//(7,95) Przesuwanie formatek sprzed 
rtfbLidSealerDrag(CLK:=P06_LidSealer.fbLidSealerDragStation.eRunningState = E_DragStationState.eDraging AND P06_LidSealer.fbLidSealerDragStation.lrActualDragPosition>80);
IF rtfbLidSealerDrag.Q THEN
	eLidSealerPackageState[1]			:=	eBeforeLidSealerPackageState[1];
	eBeforeLidSealerPackageState[1]		:=	eClearPackageState;
	eLidSealerPackageState[2]			:=	eBeforeLidSealerPackageState[2];
	eBeforeLidSealerPackageState[2]		:=	eClearPackageState;
END_IF
		
//(7,96) 
fbIbLidFeederAfterSensor 	(bIN:= 	IbLidFeederAfterSensor ,	tFilterTimeOn:=T#40MS,	tFilterTimeOff:=T#20MS); //BYŁO 20ms
ftfbIbLidFeederAfterSensor	(CLK:=	fbIbLidFeederAfterSensor.bOUT);
rtfbIbLidFeederAfterSensor	(CLK:=	fbIbLidFeederAfterSensor.bOUT);
fbMRAfterLidFeederPackageState(
						bFirstCycle:= GVL.bFirstCycle,
						bTrigger:=ftfbIbLidFeederAfterSensor.Q,
						tTriggerFilterTimeOn:=T#0MS,
						tTriggerFilterTimeOff:=T#0MS,
						bTriggerBottle:=FALSE,
						bWithBottleControl:=FALSE,
						bWithCapControl:=FALSE,
						bWithFormControlTrigerCounter:=FALSE,
						bMoveOnlyToLastExitRegister:=FALSE,
						bRotateEntranceRegisterBefore:=FALSE,
						bNoKeepTryingMove:=TRUE,
						bTriggerCap:=FALSE,
						bReset:=bResetStates,
						iEntranceArrayElements:=2,
						iExitArrayElements:=2,
						bInvertWriting:=FALSE,
						eClearPackageState:=eClearPackageState,
						bTriggerCounter:=bMRCapCorrect,
						eEntranceState:=eAfterLidFeederPackageState,
						eExitState:=eBeforeLidSealerPackageState,
						bKeepTryingMove:=bKeepTryingMove796,
						bError=>,
						iError=>,
						bTriggerDone=>,
						bTriggerFilteredOUT=>);			

// (7,97) Przesuwanie formatek spod zakrecearek za zakrecarki  
rtfbLidFeederDrag(CLK:=
						(P06_LidFeeder.fbLidFeederDragStation.eRunningState = E_DragStationState.eDraging AND P06_LidFeeder.fbLidFeederDragStation.lrActualDragPosition>80) OR
						(P06_WickFeeder.fbWickFeederDragStation.eRunningState = E_DragStationState.eDraging AND P06_WickFeeder.fbWickFeederDragStation.lrActualDragPosition>80)
						);
IF rtfbLidFeederDrag.Q THEN
	eAfterLidFeederPackageState[1]		:=	eLidFeederPackageState[1];
	eAfterLidFeederPackageState[2]		:=	eLidFeederPackageState[2];
	eLidFeederPackageState[1]			:=	eClearPackageState;
	eLidFeederPackageState[2]			:=	eClearPackageState;
END_IF

//(7,98) Przesuwanie formatek sprzed sprawdzania platynek na platynki
IF rtfbLidFeederDrag.Q THEN
	eLidFeederPackageState[1]			:=	eBeforeLidFeederPackageState[1];
	eBeforeLidFeederPackageState[1]		:=	eClearPackageState;
	eLidFeederPackageState[2]			:=	eBeforeLidFeederPackageState[2];
	eBeforeLidFeederPackageState[2]		:=	eClearPackageState;
END_IF

//(7,99)
fbIbLidFeederThirdFormSensor				(bIN:= 	IbLidFeederThirdFormSensor,					tFilterTimeOn:=T#30MS,	tFilterTimeOff:=T#30MS); 
ftfbIbLidFeederThirdFormSensor				(CLK:=	fbIbLidFeederThirdFormSensor.bOUT, 			Q=>); 
rtfbIbLidFeederThirdFormSensor				(CLK:=	fbIbLidFeederThirdFormSensor.bOUT, 			Q=>);
ftbMRBeforeLidFeeder2Block					(CLK:=	bMRBeforeLidFeeder2Block,					Q=>);
tofftbMRBeforeLidFeeder2Block				(IN:=	ftbMRBeforeLidFeeder2Block.Q,				PT:=T#1100MS);	
// Ustawianie blokady dla ruchu tylko w jedną stronę siłownika
IF ((P06_LidFeeder.fbLidFeederDragStation.eRunningState = E_DragStationState.eDraging)OR (P06_WickFeeder.fbWickFeederDragStation.eRunningState = E_DragStationState.eDraging))
	AND NOT bMRBeforeLidFeeder2Block AND NOT tofftbMRBeforeLidFeeder2Block.Q THEN
	bMRBeforeLidFeeder2Block := TRUE;
END_IF
IF bMRBeforeLidFeeder2Block AND 
	(
	(P06_LidFeeder.fbLidFeederDragStation.eRunningState = E_DragStationState.eDraging AND P06_LidFeeder.fbLidFeederDragStation.lrActualDragPosition>90) OR
	(P06_WickFeeder.fbWickFeederDragStation.eRunningState = E_DragStationState.eDraging AND P06_WickFeeder.fbWickFeederDragStation.lrActualDragPosition>90)
	)
 THEN	
	bMRBeforeLidFeeder2Block := FALSE;
END_IF

fbMRBeforeLidFeeder2PackageState(
                        bFirstCycle:= GVL.bFirstCycle,
                        bTrigger:=rtfbIbLidFeederThirdFormSensor.Q AND NOT bMRBeforeLidFeeder2Block,
                        tTriggerFilterTimeOn:=T#0MS,
                        tTriggerFilterTimeOff:=T#0MS,
                        bTriggerBottle:=FALSE,
                        bWithBottleControl:=FALSE,
                        bWithCapControl:=FALSE,
                        bWithFormControlTrigerCounter:=FALSE,
                        bRotateEntranceRegisterBefore:=FALSE,
                        bNoKeepTryingMove:=TRUE,
                        bTriggerCap:=,
                        bReset:=bResetStates,
                        iEntranceArrayElements:=4,
                        iExitArrayElements:=2,
                        bInvertWriting:=FALSE,
                        eClearPackageState:=eClearPackageState,
                        bTriggerCounter:=bMRLidFeederFormInCap,
                        eEntranceState:=eBeforeLidFeeder2PackageState,
                        eExitState:=eBeforeLidFeederPackageState,
                        bKeepTryingMove:=bKeepTryingMove799,
                        bError=>,
                        iError=>,
                        bTriggerDone=>,
                        bTriggerFilteredOUT=>); 
IF fbMRBeforeLidFeeder2PackageState.bTrigger THEN iLFTest1:=iLFTest1+1; END_IF 
// (7,99) A - Dodatkowe przesuniecie na zboczne narastajace
//IF rtfbIbLidFeederThirdFormSensor.Q AND NOT eBeforeLidFeeder2PackageState[1].bFormPresent THEN
//	eBeforeLidFeeder2PackageState[1] := eBeforeLidFeeder2PackageState[2];
//	eBeforeLidFeeder2PackageState[2] := eClearPackageState;
//	eBeforeLidFeeder2PackageState[2] := eBeforeLidFeeder2PackageState[3];
//	eBeforeLidFeeder2PackageState[3] := eClearPackageState;	
//	eBeforeLidFeeder2PackageState[3] := eBeforeLidFeeder2PackageState[4];
//	eBeforeLidFeeder2PackageState[4] := eClearPackageState;			
//END_IF


// (8) Przesuwanie formatek z wagi w kosmos	LidFeeder		
fbIbWeight1FormSensor			(bIN:= 	P05_Weight.IbWeight1FormSensor,		tFilterTimeOn:=T#40MS,	tFilterTimeOff:=T#40MS);
ftfbIbWeight1FormSensor			(CLK:=	fbIbWeight1FormSensor.bOUT, 		Q=>);	

fbMRAfterWeightPackageStateLF(		///ZMIANAAAA
						bFirstCycle:= GVL.bFirstCycle,
						bTrigger:=ftfbIbWeight1FormSensor.Q,
						tTriggerFilterTimeOn:=T#0MS,
						tTriggerFilterTimeOff:=T#0MS,
						bTriggerBottle:=FALSE,
						bWithBottleControl:=FALSE,
						bWithCapControl:=FALSE,
						bWithFormControlTrigerCounter:=FALSE,
						bMoveOnlyToLastExitRegister:=FALSE,
						bRotateEntranceRegisterBefore:=FALSE,
						bNoKeepTryingMove:=FALSE,
						bTriggerCap:=FALSE,
						bReset:=bResetStates,
						iEntranceArrayElements:=4,
						iExitArrayElements:=4,
						bInvertWriting:=FALSE,
						eClearPackageState:=eClearPackageState,
						bTriggerCounter:=bMRFormExitWeight,
						eEntranceState:=eWeightPackageState,
						eExitState:=eBeforeLidFeeder2PackageState,
						bKeepTryingMove:=bKeepTryingMove4,
						bError=>,
						iError=>,
						bTriggerDone=>,
						bTriggerFilteredOUT=>);				
											
						
// (9) Przesuwanie formatek zza dozownikow na wage
fbIbWeight4FormSensor			(bIN:= 	P05_Weight.IbWeight4FormSensor,		tFilterTimeOn:=T#40MS,	tFilterTimeOff:=T#40MS); //BYLO 20 I 20
//fbIbWeight4FormSensor			(bIN:= 	P00_ReadRFIDCard.bReadedCardAfterDispencers,		tFilterTimeOn:=T#40MS,	tFilterTimeOff:=T#40MS); //BYLO 20 I 20
ftIbWeight4FormSensor			(CLK:=	fbIbWeight4FormSensor.bOUT, 		Q=>);	
fbMRWeightPackageState(
						bFirstCycle:= GVL.bFirstCycle,
						bTrigger:=fbIbWeight4FormSensor.bOUT,//P05_Weight.IbWeight4FormSensor, 
						tTriggerFilterTimeOn:=T#100MS,
						tTriggerFilterTimeOff:=T#20MS,
						bTriggerBottle:=FALSE,
						bWithBottleControl:=FALSE,
						bWithCapControl:=FALSE,
						bWithFormControlTrigerCounter:=FALSE,
						bMoveOnlyToLastExitRegister:=FALSE,
						bRotateEntranceRegisterBefore:=FALSE,
						bNoKeepTryingMove:=FALSE,
						bTriggerCap:=FALSE,
						bReset:=bResetStates,
						iEntranceArrayElements:=4,
						iExitArrayElements:=4,
						bInvertWriting:=FALSE,
						eClearPackageState:=eClearPackageState,
						bTriggerCounter:=bTemp,
						eEntranceState:=eAfterDispencersPackageState,
						eExitState:=eWeightPackageState,
						bKeepTryingMove:=bKeepTryingMove5,
						bError=>,
						iError=>,
						bTriggerDone=>,
						bTriggerFilteredOUT=>);		

						
// (10) Przesuwanie z dozownikow za dozowniki
fbMRAfterDispencerPackageState(
						bFirstCycle:= GVL.bFirstCycle,
						//bTrigger:=P02_Dispencers.fbDispencersDragRightStation.lrActualDragPosition>=130,
						bTrigger:=P00_PackML.tonDispencersDragLeftMiddleSensor.Q, {warning 'Przeciaganie - TON zamiast pozycji'}
						tTriggerFilterTimeOn:=T#0MS,
						tTriggerFilterTimeOff:=T#0MS,
						bInvertWriting:=FALSE,
						bTriggerBottle:=FALSE,
						iEntrenceArrayElements:=4,
						iExitArrayElements:=4,
						bWithFormControlTrigerCounter:=FALSE,
						bMoveOnlyIfFormPresent:=FALSE,
						bMoveOnlyToLastExitRegister:=FALSE,
						bMoveOnlyToLastRegister:=FALSE,
						bNoKeepTryingMove:=FALSE,
						bReset:=bResetStates,
						eClearPackageState:=eClearPackageState,
						bRotateEntranceRegisterBefore:=FALSE,
						bTriggerCounter:=bMRFormExitDispencer,
						eEntranceState:=eDispencersPackageState,
						eExitState:=eAfterDispencersPackageState,
						bKeepTryingMove:=bKeepTryingMove6,
						bError=>,
						iError=>,
						bTriggerDone=>,
						bTriggerFilteredOUT=>);	

// (11) Przesuwanie sprzed dozownikow na dozowniki
fbMRDispencerPackageState(
						bFirstCycle:= GVL.bFirstCycle,
						//bTrigger:=P02_Dispencers.fbDispencersDragRightStation.lrActualDragPosition>=130,
						bTrigger:=P00_PackML.tonDispencersDragLeftMiddleSensor.Q, {warning 'Przeciaganie - TON zamiast pozycji'}						
						tTriggerFilterTimeOn:=T#0MS,
						tTriggerFilterTimeOff:=T#0MS,
						bInvertWriting:=FALSE,
						bTriggerBottle:=FALSE,
						iEntrenceArrayElements:=4,
						iExitArrayElements:=4,
						bWithFormControlTrigerCounter:=FALSE,
						bMoveOnlyIfFormPresent:=FALSE,
						bMoveOnlyToLastExitRegister:=FALSE,
						bMoveOnlyToLastRegister:=FALSE,
						bNoKeepTryingMove:=FALSE,
						bReset:=bResetStates,
						eClearPackageState:=eClearPackageState,
						bRotateEntranceRegisterBefore:=FALSE,
						bTriggerCounter:=bMRFormDispencer,
						eEntranceState:=eBeforeDispencersPackageState,
						eExitState:=eDispencersPackageState,
						bKeepTryingMove:=bKeepTryingMove7,
						bError=>,
						iError=>,
						bTriggerDone=>,
						bTriggerFilteredOUT=>);		
					
// (12) Przesuwanie formatek sprzed szlabanu rpzed dozowniki

fbFilteredFormsSensorGate(bIn:=IbFormCheckFormSensor,	tFilterTimeOn:=T#30MS,	tFilterTimeOff:=T#20MS);					
fbMRBeforeDispencersPackageStateNew(
						bFirstCycle:= GVL.bFirstCycle,
						{warning ''}
						bTrigger:=(*fbFilteredFormsSensorGate.bOUT*)bFormatSensor,
						tTriggerFilterTimeOn:=T#0MS,
						tTriggerFilterTimeOff:=T#0MS,
						{warning 'Add filtered value 2023/06/16'}
						bTriggerBottle:=bBottleSensor (*MAIN.IbBottleInFormCheckBottleSensor*) OR VIS.bSimulation,
						bWithBottleControl:=TRUE,
						bWithCapControl:=FALSE,
						bWithFormControlTrigerCounter:=FALSE,
						bMoveOnlyToLastExitRegister:=FALSE,
						bRotateEntranceRegisterBefore:=FALSE,
						bNoKeepTryingMove:=TRUE,
						bTriggerCap:=,
						bReset:=bResetStates,
						iEntranceArrayElements:=1,
						iExitArrayElements:=4,
						bInvertWriting:=FALSE,
						eClearPackageState:=eClearPackageState,
						bTriggerCounter:=bMRFormExitGate1,
						eEntranceState:=eBeforeGatePackageState,
						eExitState:=eBeforeDispencersPackageState,
						bKeepTryingMove:=bKeepTryingMove8,
						bError=>,
						iError=>,
						bTriggerDone=>,
						bTriggerFilteredOUT=>);			
	
// Przesuwanie formatek spod podjanika butelek w kosmos
eTempState2[1]:=eClearPackageState;
eTempState2[2]:=eClearPackageState;
eTempState2[3]:=eClearPackageState;
fbIbBottleFeederFormPresent(bIn:=P01_BottleFeeder.IbBottleFeederFormGateBeforeSensor,	tFilterTimeOn:=T#20MS,	tFilterTimeOff:=T#20MS);					
ftfbIbBottleFeederFormPresent(CLK:=fbIbBottleFeederFormPresent.bOUT);
				
aSetIDBottle();						
						
//Pierwszy cykl, zeby na poczatek nie wykrywalo zbocza opadajacego				
bFirstCycle:=TRUE;		
GVL.bResetStates:=FALSE;


(**** Zapisywanie RFID  ***)

a2RFID();

(**** Koniec zapisywania RFID  ***)
END_ACTION

ACTION aCycleRegister2Phase:
eClearPackageState.nID := 0;
eClearPackageState.nCardNumber:=0;
eClearPackageState.bFormPresent := FALSE;
eClearPackageState.bBottlePresent := FALSE;
eClearPackageState.bDosingTwoPhases := FALSE;
eClearPackageState.nDispencerNr := 0;
eClearPackageState.nDispencerNrSecondPhase := 0;
eClearPackageState.tDispencingTime := T#0MS;
eClearPackageState.tDispencingTimeSecondPhase := T#0MS;
eClearPackageState.lrDoseVolumeSV := 0.0;
eClearPackageState.lrDoseVolumeCV := 0.0;
eClearPackageState.lrDoseVolumeSVSecondPhase := 0.0;
eClearPackageState.lrDoseVolumeCVSecondPhase := 0.0;
eClearPackageState.bDoseAborted := FALSE;
eClearPackageState.bWeighed := FALSE;
eClearPackageState.bWeightAborted:=FALSE;
eClearPackageState.lrWeightSV := 0.0;
eClearPackageState.lrWeightCV := 0.0;
eClearPackageState.lrWeightMeasuredCV := 0.0;
eClearPackageState.lrMinWeightCV:=0.0;
eClearPackageState.lrMaxWeightCV:=0.0;	
eClearPackageState.lrWeightDif:=0.0;			
eClearPackageState.bWeightOK := FALSE;
eClearPackageState.tWeightingTime := T#0MS;
eClearPackageState.bCapPutted := FALSE;
eClearPackageState.bCapChecked := FALSE;
eClearPackageState.bCapOK := FALSE;
eClearPackageState.bCapGripperScrewed := FALSE;
eClearPackageState.bCapGripperScrewAborted := FALSE;
eClearPackageState.tCapGripperScrewingTime := T#0MS;
eClearPackageState.bCapCorrectPutted := FALSE;
eClearPackageState.bCapCorrectChecked := FALSE;
eClearPackageState.bCapCorrectNOK := FALSE;
eClearPackageState.bCapCorrectCapOn:=FALSE;
eClearPackageState.bBottleTransferedToExit := FALSE;
eClearPackageState.bBottleTransferedToLabeler := FALSE;
bAlwaysFalse:=FALSE;

// (1) HISTORIA
fbIbFirstFormCheckFormSensor	(bIN:= 	P13_BottleTransfer.IbFirstFormCheckFormSensor,	tFilterTimeOn:=T#30MS,	tFilterTimeOff:=T#30MS);// bylo 80 i 20
ftfbIbFirstFormCheckFormSensor	(CLK:=	fbIbFirstFormCheckFormSensor.bOUT, 				Q=>);
rtfbIbFirstFormCheckFormSensor	(CLK:=	fbIbFirstFormCheckFormSensor.bOUT,				Q=>);
fbIbSecondFormCheckFormSensor	(bIN:= 	P13_BottleTransfer.IbSecondFormCheckFormSensor,	tFilterTimeOn:=T#30MS,	tFilterTimeOff:=T#30MS);
rtfbIbSecondFormCheckFormSensor	(CLK:=	fbIbSecondFormCheckFormSensor.bOUT, 			Q=>);
ftfbIbSecondFormCheckFormSensor	(CLK:=	fbIbSecondFormCheckFormSensor.bOUT, 			Q=>);


// (0) Kasowanie formatek za robotem
// BOOL ustawiany przy nastepnym ruchu robota
bRFIDClearAfterRobot;					
iRFIDClearNr1AfterRobot;	
iRFIDClearNr2AfterRobot;
rtiBottleTransferCase2(CLK:=P00_PackML.iBottleTransferCase	=	2,		Q=>);
IF	rtiBottleTransferCase2.Q	THEN
	IF P00_PackML.nCounterFormsToLoad = 2 THEN
		iRFIDClearNr1AfterRobot	:=	ULINT_TO_INT(eRobotPackageState[1].nCardNumber);
		iRFIDClearNr2AfterRobot	:=	ULINT_TO_INT(eRobotPackageState[2].nCardNumber);		
	ELSIF P00_PackML.nCounterFormsToLoad = 1 THEN
		iRFIDClearNr1AfterRobot	:=	ULINT_TO_INT(eRobotPackageState[1].nCardNumber);
		iRFIDClearNr2AfterRobot	:=	0;	
	END_IF
END_IF
IF bRFIDClearAfterRobot THEN 
	FOR i:=1 TO 100 DO	
		IF iRFIDClearNr1AfterRobot > 0 THEN	{warning 'tutaj zmienić na dwa FORy i EXITy'}
			IF eRFID[i].nCardNumber = INT_TO_ULINT(iRFIDClearNr1AfterRobot) THEN
				eRFID[i]						:=	eClearPackageState;
				eRFID[i].bFormPresent			:= TRUE; // wprowadzona zmiana do testów 
				iRFIDClearNr1AfterRobot			:= 0;
				iRFIDClearNr1AfterRobotCount	:=	iRFIDClearNr1AfterRobotCount	+	1;
			END_IF
		END_IF
		IF iRFIDClearNr2AfterRobot > 0 THEN
			IF eRFID[i].nCardNumber = INT_TO_ULINT(iRFIDClearNr2AfterRobot) THEN
				eRFID[i]						:=	eClearPackageState;
				eRFID[i].bFormPresent			:= TRUE;  // Wprowadzona zmiana do testów
				iRFIDClearNr2AfterRobot			:= 0;
				
				iRFIDClearNr2AfterRobotCount	:=	iRFIDClearNr2AfterRobotCount	+	1;
			END_IF
		END_IF		
		IF 	iRFIDClearNr1AfterRobot = 0 AND iRFIDClearNr2AfterRobot = 0 THEN
			bRFIDClearAfterRobot	:=	FALSE;
		END_IF
	END_FOR;
END_IF



IF ftfbIbFirstFormCheckFormSensor.Q THEN
	
	FOR i := 999 TO 2 BY -1 DO		
		eHistoryPackageState[i] := eHistoryPackageState[i-1];
	END_FOR		
	
	FOR i:=1 TO 100 DO	
	
		IF eRobotPackageState[1].nCardNumber=eRFID[i].nCardNumber THEN
			eRFID[i]		:=	eRobotPackageState[1];
			EXIT;
		END_IF;
	
	END_FOR;
	
	eHistoryPackageState[1]	:=	eRobotPackageState[1];
	eRobotPackageState[1]	:=	eClearPackageState; // dodane na testy
	nCheckRobotDone			:=	nCheckRobotDone+1;
	
END_IF

IF bResetStates THEN
	eRobotPackageState[1]:=eClearPackageState;
	eRobotPackageState[2]:=eClearPackageState;
	eRobotTempState[1]:=eClearPackageState;// dodane na testy 31.05
END_IF

IF nFormCounter = 1000 OR bResetHistory THEN 
	FOR i := 1 TO 1000 DO
		eHistoryPackageState[i]:=eClearPackageState;
	END_FOR
	
	nFormCounter := 0 ;
	nID := 0;
END_IF


// (2) PRZESUWANIE POD ROBOTEM
IF rtfbIbFirstFormCheckFormSensor.Q THEN
	eRobotPackageState[1]				:= eRobotTempState[1];
	eRobotTempState[1]					:= eClearPackageState;
END_IF

IF  ftfbIbSecondFormCheckFormSensor.Q THEN
	eRobotTempState[1]					:=	eRobotPackageState[2];
	eRobotPackageState[2]				:=	eClearPackageState;
END_IF

IF rtfbIbSecondFormCheckFormSensor.Q THEN
	eRobotPackageState[2].bFormPresent	:=	TRUE;
END_IF

// (3) Przesuwanie formatek zza zakrecarek pod sprwadzanie nakretek
//Przesuwanie formatek spod sprawdzania zakretek na robota
//Usuwanie rejestru bo jest nieuzywant	
//eUnderCorrectCapPackageState[1]			:=	eClearPackageState;	
eUnderCorrectCapPackageState[2]			:=	eClearPackageState;	
eUnderCorrectCapPackageState[3]			:=	eClearPackageState;	
eUnderCorrectCapPackageState[4]			:=	eClearPackageState;	
eUnderCorrectCapPackageState[5]			:=	eClearPackageState;	
eUnderCorrectCapPackageState[6]			:=	eClearPackageState;		
eUnderCorrectCapPackageState[7]			:=	eClearPackageState;		
eUnderCorrectCapPackageState[8]			:=	eClearPackageState;									//bylo 400ms?
fbIbCapCorrectCheckFormSensor			(bIN:= 	P11_CapCorrectCheck.IbCapCorrectCheckFormSensor,	tFilterTimeOn:=T#10MS,	tFilterTimeOff:=T#0MS); //BYŁO 20ms
rtfbIbCapCorrectCheckFormSensor			(CLK:=	fbIbCapCorrectCheckFormSensor.bOUT, 					Q=>); // dd do testów
ftfbIbCapCorrectCheckFormSensor			(CLK:=	fbIbCapCorrectCheckFormSensor.bOUT, 					Q=>);

//Czujnik przesuwania rejestru za zakręcarką
fbIbCapCorrectCheckAfterScrewerFormSensor (bIN:= 	P11_CapCorrectCheck.IbCapCorrectCheckAfterScrewerFormSensor,	tFilterTimeOn:=T#40MS,	tFilterTimeOff:=T#0MS); //BYŁO 20ms
ftfbIbCapCorrectCheckAfterScrewerFormSensor(CLK:=fbIbCapCorrectCheckAfterScrewerFormSensor.bOUT);

IF rtfbIbCapCorrectCheckFormSensor.Q AND NOT eUnderCorrectCapPackageState[1].bFormPresent THEN  			//dd do testów USUNAĆ
	eUnderCorrectCapPackageState[1].bFormPresent  :=	TRUE;  												//dd do testów USUNAĆ
	iTestCCC2	:=	iTestCCC2	+	1;																		//dd do testów USUNAĆ
END_IF  																								

IF 	ftfbIbCapCorrectCheckFormSensor.Q THEN
	eUnderCorrectCapPackageState[1]	:=	eClearPackageState;
	iTestCCC1	:=	iTestCCC1	+	1;
END_IF

fbMRCorrectCapPackageState(
						bFirstCycle:= GVL.bFirstCycle,
						bTrigger:=(*ftfbIbCapCorrectCheckFormSensor.Q*)ftfbIbCapCorrectCheckAfterScrewerFormSensor.Q,
						tTriggerFilterTimeOn:=T#0MS,
						tTriggerFilterTimeOff:=T#0MS,
						bTriggerBottle:=FALSE,
						bWithBottleControl:=FALSE,
						bWithCapControl:=FALSE,
						bWithFormControlTrigerCounter:=FALSE,
						bMoveOnlyToLastExitRegister:=FALSE,
						bRotateEntranceRegisterBefore:=FALSE,
						bNoKeepTryingMove:=TRUE,
						bTriggerCap:=FALSE,
						bReset:=bResetStates,
						iEntranceArrayElements:=2,
						iExitArrayElements:=8,
						bInvertWriting:=FALSE,
						eClearPackageState:=eClearPackageState,
						bTriggerCounter:=bMRCapCorrect,
						eEntranceState:=eAfterScrewerPackageState,
						//eExitState:=eUnderCorrectCapPackageState, //dd do testów USUNAĆ
						eExitState:=eUnderCorrectCapPackageStateTemp,						
						bKeepTryingMove:=bKeepTryingMove1,
						bError=>,
						iError=>,
						bTriggerDone=>,
						bTriggerFilteredOUT=>);			

eUnderCorrectCapPackageStateTemp[1]:= eClearPackageState; //dd do testów USUNAĆ
eUnderCorrectCapPackageStateTemp[2]:= eClearPackageState;//dd do testów USUNAĆ 
						
// (4) Przesuwanie formatek spod zakrecearek za zakrecarki  
//rtfbFormsDragingPneumaticStationDragging(CLK:=P10_GripperScrewer.fbGripperScrewersDragStation.eRunningState = E_DragStationState.eDraging);
rtfbFormsDragingPneumaticStationDragging(CLK:=P10_GripperScrewer.fbGripperScrewersDragStation.eRunningState = E_DragStationState.eDraging AND P10_GripperScrewer.fbGripperScrewersDragStation.lrActualDragPosition>80);

IF rtfbFormsDragingPneumaticStationDragging.Q THEN
	eAfterScrewerPackageState[1]		:=	eUnderScrewerPackageState[1];
	eAfterScrewerPackageState[2]		:=	eUnderScrewerPackageState[2];
	eUnderScrewerPackageState[1]		:=	eClearPackageState;
	eUnderScrewerPackageState[2]		:=	eClearPackageState;
END_IF

								
// (5) Przesuwanie formatek sprzed zakrecarek na zakrecarki
IF rtfbFormsDragingPneumaticStationDragging.Q THEN
	eUnderScrewerPackageState[1]		:=	eBeforeScrewersPackageState[1];
	eBeforeScrewersPackageState[1]		:=	eClearPackageState;
	eUnderScrewerPackageState[2]		:=	eBeforeScrewers2PackageState[1];
	eBeforeScrewers2PackageState[1]		:=	eClearPackageState;
END_IF

// (6) Przesuwanie formatek zza sprawdzania zalozenia na przed zakrecarki
fbIbScrewerThirdFormCheckFormSensor			(bIN:= 	P10_GripperScrewer.IbGripperScrewersThirdFormCheckFormSensor,		tFilterTimeOn:=T#30MS,	tFilterTimeOff:=T#30MS); //BYŁO 20ms
ftfbIbScrewerThirdFormCheckFormSensor		(CLK:=	fbIbScrewerThirdFormCheckFormSensor.bOUT, 			Q=>);
rtfbIbScrewerThirdFormCheckFormSensor		(CLK:=	fbIbScrewerThirdFormCheckFormSensor.bOUT, 			Q=>);
bTrendIbThirdFormCheckFormSensor:=P10_GripperScrewer.IbGripperScrewersThirdFormCheckFormSensor;
bTrendFilteredIbThirdFormCheckFormSensor:=ftfbIbScrewerThirdFormCheckFormSensor.Q;
ftbMRBeforeScrewer2Block 					(CLK:=	bMRBeforeScrewer2Block,								Q=>);
tofftbMRBeforeScrewer2Block					(IN:=	ftbMRBeforeScrewer2Block.Q,							PT:=T#1100MS);//bylo 350		//  bylo 1000			


// Ustawianie blokady dla ruchu tylko w jedną stronę siłownika
IF ( P10_GripperScrewer.fbGripperScrewersDragStation.eRunningState = E_DragStationState.eDraging )
	AND NOT bMRBeforeScrewer2Block AND NOT tofftbMRBeforeScrewer2Block.Q THEN
	bMRBeforeScrewer2Block := TRUE;
END_IF

//IF bMRBeforeScrewer2Block AND P00_PackML.tonGripperScrewerDragMiddleSensor.Q THEN
IF bMRBeforeScrewer2Block AND P10_GripperScrewer.fbGripperScrewersDragStation.eRunningState = E_DragStationState.eDraging AND P10_GripperScrewer.fbGripperScrewersDragStation.lrActualDragPosition>90 THEN	
	bMRBeforeScrewer2Block := FALSE;
END_IF


//(6)
fbMRBeforeScrewer2PackageState(
                        bFirstCycle:= GVL.bFirstCycle,
                        bTrigger:=ftfbIbScrewerThirdFormCheckFormSensor.Q AND NOT bMRBeforeScrewer2Block,
                        tTriggerFilterTimeOn:=T#0MS,
                        tTriggerFilterTimeOff:=T#0MS,
                        bTriggerBottle:=FALSE,
                        bWithBottleControl:=FALSE,
                        bWithCapControl:=FALSE,
                        bWithFormControlTrigerCounter:=FALSE,
                        bRotateEntranceRegisterBefore:=FALSE,
                        bNoKeepTryingMove:=TRUE,
                        bTriggerCap:=,
                        bReset:=bResetStates,
                        iEntranceArrayElements:=2,
                        iExitArrayElements:=2,
                        bInvertWriting:=FALSE,
                        eClearPackageState:=eClearPackageState,
                        bTriggerCounter:=bMRFormInCap,
                        eEntranceState:=eBeforeScrewers2PackageState,
                        eExitState:=eBeforeScrewersPackageState,
                        bKeepTryingMove:=bKeepTryingMove2,
                        bError=>,
                        iError=>,
                        bTriggerDone=>,
                        bTriggerFilteredOUT=>);   										

// (6) A - Dodatkowe przesuniecie na zboczne narastajace
IF rtfbIbScrewerThirdFormCheckFormSensor.Q AND NOT eBeforeScrewers2PackageState[1].bFormPresent THEN
	eBeforeScrewers2PackageState[1] := eBeforeScrewers2PackageState[2];
	eBeforeScrewers2PackageState[2] := eClearPackageState;
END_IF

						
//(7) Przesuwanie formatek spod sprawdzania zalozenia na przed zakrecarki
fbIbCapPuttedCheckFormSensor		(bIN:= 	P09_CapPuttedCheck.IbCapPuttedCheckFormSensor,		tFilterTimeOn:=T#30MS,	tFilterTimeOff:=T#30MS); //Było 20ms
fbIbCapPuttedCheckFormSensorv2		(bIN:= 	P09_CapPuttedCheck.IbCapPuttedCheckFormSensor,		tFilterTimeOn:=T#30MS,	tFilterTimeOff:=T#30MS); //Było 20ms
ftfbIbCapPuttedCheckFormSensor		(CLK:=	fbIbCapPuttedCheckFormSensorv2.bOUT, 					Q=>);

IF ftfbIbCapPuttedCheckFormSensor.Q THEN
	iftfbIbCapPuttedCheckFormSensor := iftfbIbCapPuttedCheckFormSensor+1;
END_IF


bBitTestOn:=TRUE;


fbMRBeforeScrewerPackageState(
                        bFirstCycle:= GVL.bFirstCycle,
                        bTrigger:=ftfbIbCapPuttedCheckFormSensor.Q,
                        tTriggerFilterTimeOn:=T#0MS,
                        tTriggerFilterTimeOff:=T#0MS,
                        bWithCapControl:=TRUE,
                      	bNoKeepTryingMove:=TRUE,
                        bTriggerCap:=P09_CapPuttedCheck.eCapPuttedCheckRunningState = E_CheckerState.eCapOK,
                        bReset:=bResetStates,
                        iEntranceArrayElements:=1,
                        iExitArrayElements:=2,
                        eClearPackageState:=eClearPackageState,
                        eEntranceState:=eBeforeCapControlPackageState,
                        eExitState:=eBeforeScrewers2PackageState,
                        bKeepTryingMove:=bKeepTryingMove3,
						bRFIDReaded:=bRFIDSBeforeScrewerWriteToRegister, // Ustawiany jeżeli Dane z tablicy RFID zostały wpisane do zwykłego rejestru
                        iBottleWithoutCap:=iCapFeederCheckCountNOK,
                        bError=>,
                        iError=>,
                        bTriggerDone=>,
                        bTriggerFilteredOUT=>);   


						
// --------------------------------------

aCycleRegisterROPP();

// (7,5-7,9) Przesuwanie pod sorterem nasadek

aCycleRegisterCapSorter();

// --------------------------------------						
						
// (8) Przesuwanie formatek z wagi w kosmos	

eTempState1[1]:=eClearPackageState;
eTempState1[2]:=eClearPackageState;
eTempState1[3]:=eClearPackageState;
fbIbWeight5FormSensor			(bIN:= 	P05_Weight.IbWeight5FormSensor,		tFilterTimeOn:=T#20MS,	tFilterTimeOff:=T#20MS);
ftfbIbWeight5FormSensor			(CLK:=	fbIbWeight5FormSensor.bOUT, 		Q=>);		
fbMRAfterWeightPackageState(
						bFirstCycle:= GVL.bFirstCycle,
						bTrigger:=ftfbIbWeight5FormSensor.Q,
						tTriggerFilterTimeOn:=T#0MS,
						tTriggerFilterTimeOff:=T#0MS,
						bTriggerBottle:=FALSE,
						bWithBottleControl:=FALSE,
						bWithCapControl:=FALSE,
						bWithFormControlTrigerCounter:=FALSE,
						bMoveOnlyToLastExitRegister:=FALSE,
						bRotateEntranceRegisterBefore:=FALSE,
						bNoKeepTryingMove:=FALSE,
						bTriggerCap:=FALSE,
						bReset:=bResetStates,
						iEntranceArrayElements:=2,
						iExitArrayElements:=4,
						bInvertWriting:=FALSE,
						eClearPackageState:=eClearPackageState,
						bTriggerCounter:=bMRFormExitWeight,
						eEntranceState:=eWeightPackage2PhasePackageState,
						eExitState:=eTempState1,
						bKeepTryingMove:=bKeepTryingMove4,
						bError=>,
						iError=>,
						bTriggerDone=>,
						bTriggerFilteredOUT=>);				

// Przesuwanie formatek dozowników na wagę

fbIbWeight6FormSensor			(bIN:= 	P05_Weight.IbWeight6FormSensor,		tFilterTimeOn:=T#20MS,	tFilterTimeOff:=T#20MS);
ftIbWeight6FormSensor			(CLK:=	fbIbWeight6FormSensor.bOUT, 		Q=>);	
fbMRWeight2PhasePackageState(
						bFirstCycle:= GVL.bFirstCycle,
						bTrigger:=fbIbWeight6FormSensor.bOUT,//P05_Weight.IbWeight6FormSensor, 
						tTriggerFilterTimeOn:=T#100MS,//bylo 50 
						tTriggerFilterTimeOff:=T#20MS,
						bTriggerBottle:=FALSE,
						bWithBottleControl:=FALSE,
						bWithCapControl:=FALSE,
						bWithFormControlTrigerCounter:=FALSE, //bylo true
						bMoveOnlyToLastExitRegister:=FALSE,
						bRotateEntranceRegisterBefore:=FALSE,
						bNoKeepTryingMove:=FALSE,
						bTriggerCap:=FALSE,
						bReset:=bResetStates,
						iEntranceArrayElements:=2,
						iExitArrayElements:=2,
						bInvertWriting:=FALSE,
						eClearPackageState:=eClearPackageState,
						bTriggerCounter:=bTemp,
						eEntranceState:=eAfterDispencer12PackageState2Phase,
						eExitState:=eWeightPackage2PhasePackageState,
						bKeepTryingMove:=bKeepTryingMove15,
						bError=>,
						iError=>,
						bTriggerDone=>,
						bTriggerFilteredOUT=>);		

//Przesuwanie formatek sprzed dozowników 12 ( pierwsze 2 z lewej strony) za dozowniki
						
fbMRAfterDispencer12PackageState(
						bFirstCycle:= GVL.bFirstCycle,
//dp					bTrigger:=P02_Dispencers.fbDispencersDragLeftStation.lrActualDragPosition<=30, // do zmiany 
						bTrigger:=P00_PackML.tonDispencersDragLeftMiddleSensor.Q,
						tTriggerFilterTimeOn:=T#0MS,
						tTriggerFilterTimeOff:=T#0MS,
						bInvertWriting:=FALSE,
						bTriggerBottle:=FALSE,
						iEntrenceArrayElements:=2,
						iExitArrayElements:=2,
						bWithFormControlTrigerCounter:=FALSE,
						bMoveOnlyIfFormPresent:=FALSE,
						bMoveOnlyToLastExitRegister:=FALSE,
						bMoveOnlyToLastRegister:=FALSE,
						bNoKeepTryingMove:=FALSE,
						bReset:=bResetStates,
						eClearPackageState:=eClearPackageState,
						bRotateEntranceRegisterBefore:=FALSE,
						bTriggerCounter:=bMRFormExitDispencer12,
						eEntranceState:=eDispencer12PackageState2Phase,
						eExitState:=eAfterDispencer12PackageState2Phase,
						bKeepTryingMove:=bKeepTryingMove6,
						bError=>,
						iError=>,
						bTriggerDone=>,
						bTriggerFilteredOUT=>);							

// Przesuwanie formatek sprzed dozowników 12 na dozowniki 12	
fbMRDispencer12PackageState(
						bFirstCycle:= GVL.bFirstCycle,
//dp					bTrigger:=P02_Dispencers.fbDispencersDragLeftStation.lrActualDragPosition<=30, // zmienic pozycje
						bTrigger:=P00_PackML.tonDispencersDragLeftMiddleSensor.Q,
						tTriggerFilterTimeOn:=T#0MS,
						tTriggerFilterTimeOff:=T#0MS,
						bInvertWriting:=FALSE,
						bTriggerBottle:=FALSE,
						iEntrenceArrayElements:=2,
						iExitArrayElements:=2,
						bWithFormControlTrigerCounter:=FALSE,
						bMoveOnlyIfFormPresent:=FALSE,
						bMoveOnlyToLastExitRegister:=FALSE,
						bMoveOnlyToLastRegister:=FALSE,
						bNoKeepTryingMove:=FALSE,
						bReset:=bResetStates,
						eClearPackageState:=eClearPackageState,
						bRotateEntranceRegisterBefore:=FALSE,
						bTriggerCounter:=bMRFormDispencer12,
						eEntranceState:=eBeforeDispencer12PackageState2Phase,
						eExitState:=eDispencer12PackageState2Phase,
						bKeepTryingMove:=bKeepTryingMove7,
						bError=>,
						iError=>,
						bTriggerDone=>,
						bTriggerFilteredOUT=>);		

//Przesuwanie formatek pomiedzy dozownikami 						
	
ftFormSensorBetweenDispencer(CLK:=fbIbFormSensorBetweenDispencer.bOUT,Q=>);
rtFormSensorBetweenDispencer(CLK:=fbIbFormSensorBetweenDispencer.bOUT,Q=>);
fbIbFormSensorBetweenDispencer(bIn:=MAIN.IbTwoPhasesFormSensorBetweenDispencers, tFilterTimeOn:=T#35MS, tFilterTimeOff:=T#35MS);



	
fbMRBetweenDispencerPackageState(
						bFirstCycle:= GVL.bFirstCycle,
						bTrigger:=rtFormSensorBetweenDispencer.Q, 
						tTriggerFilterTimeOn:=T#0MS,
						tTriggerFilterTimeOff:=T#0MS,
						bTriggerBottle:=FALSE,
						bWithBottleControl:=FALSE,
						bWithCapControl:=FALSE,
						bWithFormControlTrigerCounter:=FALSE,
						bMoveOnlyToLastExitRegister:=FALSE,
						bRotateEntranceRegisterBefore:=FALSE,
						bNoKeepTryingMove:=FALSE,
						bTriggerCap:=FALSE,
						bReset:=bResetStates,
						iEntranceArrayElements:=2,
						iExitArrayElements:=2,
						bInvertWriting:=FALSE,
						eClearPackageState:=eClearPackageState,
						bTriggerCounter:=bMRFormBetweenDispencer,
						eEntranceState:=eAfterDispencer34PackageState2Phase,
						eExitState:=eBeforeDispencer12PackageState2Phase,
						bKeepTryingMove:=bKeepTryingMove9,
						bError=>,
						iError=>,
						bTriggerDone=>,
						bTriggerFilteredOUT=>);		
					
//Przesuwanie formatek sprzed dozowników 34 ( pierwsze 2 z prawej storny ) za dozowniki
						
fbMRAfterDispencer34PackageState(
						bFirstCycle:= GVL.bFirstCycle,
//dp					bTrigger:=P02_Dispencers.fbDispencersDragRightStation.lrActualDragPosition>=135, // do zmiany 
						bTrigger:=P00_PackML.tonDispencersDragRightMiddleSensor.Q, {warning 'Przeciaganie - TON zamiast pozycji'}						
						tTriggerFilterTimeOn:=T#0MS,
						tTriggerFilterTimeOff:=T#0MS,
						bInvertWriting:=FALSE,
						bTriggerBottle:=FALSE,
						iEntrenceArrayElements:=2,
						iExitArrayElements:=2,
						bWithFormControlTrigerCounter:=FALSE,
						bMoveOnlyIfFormPresent:=FALSE,
						bMoveOnlyToLastExitRegister:=FALSE,
						bMoveOnlyToLastRegister:=FALSE,
						bNoKeepTryingMove:=FALSE,
						bReset:=bResetStates,
						eClearPackageState:=eClearPackageState,
						bRotateEntranceRegisterBefore:=FALSE,
						bTriggerCounter:=bMRFormExitDispencer34,
						eEntranceState:=eDispencer34PackageState2Phase,
						eExitState:=eAfterDispencer34PackageState2Phase,
						bKeepTryingMove:=bKeepTryingMove6,
						bError=>,
						iError=>,
						bTriggerDone=>,
						bTriggerFilteredOUT=>);							

// Przesuwanie formatek sprzed dozowników 34 na dozowniki 34	
fbMRDispencer34PackageState(
						bFirstCycle:= GVL.bFirstCycle,
//dp					bTrigger:=P02_Dispencers.fbDispencersDragRightStation.lrActualDragPosition>=135, // zmienic pozycje
						bTrigger:=P00_PackML.tonDispencersDragRightMiddleSensor.Q, {warning 'Przeciaganie - TON zamiast pozycji'}						
						tTriggerFilterTimeOn:=T#0MS,
						tTriggerFilterTimeOff:=T#0MS,
						bInvertWriting:=FALSE,
						bTriggerBottle:=FALSE,
						iEntrenceArrayElements:=2,
						iExitArrayElements:=2,
						bWithFormControlTrigerCounter:=FALSE,
						bMoveOnlyIfFormPresent:=FALSE,
						bMoveOnlyToLastExitRegister:=FALSE,
						bMoveOnlyToLastRegister:=FALSE,
						bNoKeepTryingMove:=FALSE,
						bReset:=bResetStates,
						eClearPackageState:=eClearPackageState,
						bRotateEntranceRegisterBefore:=FALSE,
						bTriggerCounter:=bMRFormDispencer34,
						eEntranceState:=eBeforeDispencer34PackageState2Phase,
						eExitState:=eDispencer34PackageState2Phase,
						bKeepTryingMove:=bKeepTryingMove7,
						bError=>,
						iError=>,
						bTriggerDone=>,
						bTriggerFilteredOUT=>);			

// Przesuwanie formatek sprzed szlabanu przed dozowniki 34
fbFilteredFormsSensorGate(bIn:=IbFormCheckFormSensor,	tFilterTimeOn:=T#20MS,	tFilterTimeOff:=T#20MS);					
						
fbMRBeforeDispencersPackageStateNew(
						bFirstCycle:= GVL.bFirstCycle,
						bTrigger:=(*fbFilteredFormsSensorGate.bOUT*)bFormatSensor,
						tTriggerFilterTimeOn:=T#0MS,
						tTriggerFilterTimeOff:=T#0MS,
						{warning 'Add filtered value 2023/06/16'}
						bTriggerBottle:= bBottleSensor (*MAIN.IbBottleInFormCheckBottleSensor*)  OR VIS.bSimulation,
						bWithBottleControl:=TRUE,
						bWithCapControl:=FALSE,
						bWithFormControlTrigerCounter:=FALSE,
						bMoveOnlyToLastExitRegister:=FALSE,
						bRotateEntranceRegisterBefore:=FALSE,
						bNoKeepTryingMove:=TRUE,
						bTriggerCap:=,
						bReset:=bResetStates,
						iEntranceArrayElements:=1,
						iExitArrayElements:=2,
						bInvertWriting:=FALSE,
						eClearPackageState:=eClearPackageState,
						bTriggerCounter:=bMRFormExitGate1,
						eEntranceState:=eBeforeGatePackageState,
						eExitState:=eBeforeDispencer34PackageState2Phase,
						bKeepTryingMove:=bKeepTryingMove8,
						bError=>,
						iError=>,
						bTriggerDone=>,
						bTriggerFilteredOUT=>);								

// Przesuwanie formatek spod podjanika butelek w kosmos

eTempState2[1]:=eClearPackageState;
eTempState2[2]:=eClearPackageState;
eTempState2[3]:=eClearPackageState;
fbIbBottleFeederFormPresent(bIn:=P01_BottleFeeder.IbBottleFeederFormGateBeforeSensor,	tFilterTimeOn:=T#20MS,	tFilterTimeOff:=T#20MS);					
ftfbIbBottleFeederFormPresent(CLK:=fbIbBottleFeederFormPresent.bOUT);
					
			
aSetIDBottle();						
	
					
//Pierwszy cykl, zeby na poczatek nie wykrywalo zbocza opadajacego				
bFirstCycle:=TRUE;		
GVL.bResetStates:=FALSE;


// Zamian rejestrów


(**** Zapisywanie RFID  ***)

a2RFID();

(**** Koniec zapisywania RFID  ***)
END_ACTION

ACTION aCycleRegisterCapSorter:

// (7,5) Przesuwanie formatek zza sortera w kosmos
//Czujnik nie mruga
tonIbCapSorterAfterFormSensor(IN:= NOT MAIN.IbCapSorterAfterFormSensor, PT:=T#1S);
IF tonIbCapSorterAfterFormSensor.Q THEN
	eAfterCapSorterPackageState[4]	:= eClearPackageState;
	eAfterCapSorterPackageState[3]	:= eClearPackageState;
	eAfterCapSorterPackageState[2]	:= eClearPackageState;
	eAfterCapSorterPackageState[1]	:= eClearPackageState;
END_IF

// (7,6) Przesuwanie z sortera nakrętek za sorter
fbMRAfterCapSorterPackageState(
						bFirstCycle:= GVL.bFirstCycle,
						bTrigger:=P00_PackML.tonCapSorterDragMiddleSensor.Q,
						tTriggerFilterTimeOn:=T#0MS,
						tTriggerFilterTimeOff:=T#0MS,
						bInvertWriting:=FALSE,
						bTriggerBottle:=FALSE,
						iEntrenceArrayElements:=4,
						iExitArrayElements:=4,
						bWithFormControlTrigerCounter:=FALSE,
						bMoveOnlyIfFormPresent:=FALSE,
						bMoveOnlyToLastExitRegister:=FALSE,
						bMoveOnlyToLastRegister:=FALSE,
						bNoKeepTryingMove:=FALSE,
						bReset:=bResetStates,
						eClearPackageState:=eClearPackageState,
						bRotateEntranceRegisterBefore:=FALSE,
						bTriggerCounter:=bTemp,
						eEntranceState:=eCapSorterPackageState,
						eExitState:=eAfterCapSorterPackageState,
						bKeepTryingMove:=bKeepTryingMove17,
						bError=>,
						iError=>,
						bTriggerDone=>,
						bTriggerFilteredOUT=>);	

// (7,7) Przesuwanie sprzed sortera na sorter
fbMRCapSorterPackageState(
						bFirstCycle:= GVL.bFirstCycle,
						bTrigger:=P00_PackML.tonCapSorterDragMiddleSensor.Q, 					
						tTriggerFilterTimeOn:=T#0MS,
						tTriggerFilterTimeOff:=T#0MS,
						bInvertWriting:=FALSE,
						bTriggerBottle:=FALSE,
						iEntrenceArrayElements:=4,
						iExitArrayElements:=4,
						bWithFormControlTrigerCounter:=FALSE,
						bMoveOnlyIfFormPresent:=FALSE,
						bMoveOnlyToLastExitRegister:=FALSE,
						bMoveOnlyToLastRegister:=FALSE,
						bNoKeepTryingMove:=FALSE,
						bReset:=bResetStates,
						eClearPackageState:=eClearPackageState,
						bRotateEntranceRegisterBefore:=FALSE,
						bTriggerCounter:=bTemp,
						eEntranceState:=eBeforeCapSorterPackageState,
						eExitState:=eCapSorterPackageState,
						bKeepTryingMove:=bKeepTryingMove18,
						bError=>,
						iError=>,
						bTriggerDone=>,
						bTriggerFilteredOUT=>);		
					
// (7,8) Przesuwanie formatek sprzed szlabanu przed sorter
fbFilteredCapSorterFormsSensorGate		(bIn:=P00_ReadRFIDCard.bReadedCardCapSorter,		tFilterTimeOn:=T#50MS,	tFilterTimeOff:=T#0MS);					
ftfbFilteredCapSorterFormsSensorGate	(CLK:=fbFilteredCapSorterFormsSensorGate.bOUT,Q=>);
fbMRBeforeCapSorterPackageState(
						bFirstCycle:= GVL.bFirstCycle,
						bTrigger:=ftfbFilteredCapSorterFormsSensorGate.Q,
						tTriggerFilterTimeOn:=T#0MS,
						tTriggerFilterTimeOff:=T#0MS,
						bTriggerBottle:=,
						bWithBottleControl:=FALSE,
						bWithCapControl:=FALSE,
						bWithFormControlTrigerCounter:=FALSE,
						bMoveOnlyToLastExitRegister:=FALSE,
						bRotateEntranceRegisterBefore:=FALSE,
						bNoKeepTryingMove:=TRUE,
						bTriggerCap:=,
						bReset:=bResetStates,
						iEntranceArrayElements:=1,
						iExitArrayElements:=4,
						bInvertWriting:=FALSE,
						eClearPackageState:=eClearPackageState,
						bTriggerCounter:=bTemp,
						eEntranceState:=eBeforeGateCapSorterPackageState,
						eExitState:=eBeforeCapSorterPackageState,
						bKeepTryingMove:=bKeepTryingMove19,
						bError=>,
						iError=>,
						bTriggerDone=>,
						bTriggerFilteredOUT=>);
END_ACTION

ACTION aCycleRegisterROPP:

eBeforeROPPCapControlPackageState;	
eBeforeROPPPackageState	;			
eBeforeROPP2PackageState	;		
eUnderROPPPackageState 		;			
eUnderROPPCorrectCapPackageState	;

// (3) Przesuwanie formatek zza zakrecarek pod sprwadzanie nakretek
IF P00_PackML.rtfbbReadedCardAfterROPP.Q AND NOT eUnderROPPCorrectCapPackageState[1].bFormPresent THEN  	
	eUnderROPPCorrectCapPackageState[1].bFormPresent		:=	TRUE;  				END_IF  																								
IF 	P00_PackML.ftfbbReadedCardAfterROPP.Q THEN
	eUnderROPPCorrectCapPackageState[1]						:=	eClearPackageState;	END_IF
				
// (4) Przesuwanie formatek spod zakrecearek za zakrecarki  
rtfbROPPDrag(CLK:=P07_ROPP.fbROPPDrag.eRunningState = E_DragStationState.eDraging AND P07_ROPP.fbROPPDrag.lrActualDragPosition>80);
IF rtfbROPPDrag.Q THEN
	eUnderROPPPackageState[1]		:=	eClearPackageState;
	eUnderROPPPackageState[2]		:=	eClearPackageState;
END_IF
						
// (5) Przesuwanie formatek sprzed zakrecarek na zakrecarki
IF rtfbROPPDrag.Q THEN
	eUnderROPPPackageState[1]		:=	eBeforeROPPPackageState[1];
	eBeforeROPPPackageState[1]		:=	eClearPackageState;
	eUnderROPPPackageState[2]		:=	eBeforeROPP2PackageState[1];
	eBeforeROPP2PackageState[1]		:=	eClearPackageState;
END_IF

// (6) Przesuwanie formatek zza sprawdzania zalozenia na przed zakrecarki
ftbMRBeforeROPP2Block 						(CLK:=	bMRBeforeROPP2Block,								Q=>);
tofftbMRBeforeROPP2Block					(IN:=	ftbMRBeforeROPP2Block.Q,							PT:=T#1100MS);	

// Ustawianie blokady dla ruchu tylko w jedną stronę siłownika
IF P07_ROPP.fbROPPDrag.eRunningState = E_DragStationState.eDraging 
	AND NOT bMRBeforeROPP2Block AND NOT tofftbMRBeforeScrewer2Block.Q THEN
	bMRBeforeROPP2Block := TRUE;
END_IF

IF bMRBeforeROPP2Block AND P07_ROPP.fbROPPDrag.eRunningState = E_DragStationState.eDraging AND P07_ROPP.fbROPPDrag.lrActualDragPosition>90 THEN	
	bMRBeforeROPP2Block := FALSE;
END_IF

//(6)
fbMRBeforeROPP2PackageState(
                        bFirstCycle:= GVL.bFirstCycle,
                        bTrigger:=P00_PackML.ftfbIbROPPThirdFormSensor.Q AND NOT bMRBeforeROPP2Block,
                        tTriggerFilterTimeOn:=T#0MS,
                        tTriggerFilterTimeOff:=T#0MS,
                        bTriggerBottle:=FALSE,
                        bWithBottleControl:=FALSE,
                        bWithCapControl:=FALSE,
                        bWithFormControlTrigerCounter:=FALSE,
                        bRotateEntranceRegisterBefore:=FALSE,
                        bNoKeepTryingMove:=TRUE,
                        bTriggerCap:=,
                        bReset:=bResetStates,
                        iEntranceArrayElements:=3,
                        iExitArrayElements:=2,
                        bInvertWriting:=FALSE,
                        eClearPackageState:=eClearPackageState,
                        bTriggerCounter:=bROPPMR,
                        eEntranceState:=eBeforeROPP2PackageState,
                        eExitState:=eBeforeROPPPackageState,
                        bKeepTryingMove:=bKeepTryingMoveROPP1,
                        bError=>,
                        iError=>,
                        bTriggerDone=>,
                        bTriggerFilteredOUT=>);   										

// (6) A - Dodatkowe przesuniecie na zboczne narastajace
IF P00_PackML.rtfbIbROPPThirdFormSensor.Q AND NOT eBeforeROPP2PackageState[1].bFormPresent THEN
	eBeforeROPP2PackageState[1] := eBeforeROPP2PackageState[2];
	eBeforeROPP2PackageState[2] := eBeforeROPP2PackageState[3];
	eBeforeROPP2PackageState[3] := eClearPackageState;
END_IF
					
//(7) Przesuwanie formatek spod sprawdzania zalozenia na przed zakrecarki
fbMRBeforeROPPPackageState(
                        bFirstCycle:= GVL.bFirstCycle,
                        bTrigger:= P00_PackML.ftbReadedCardBeforeROPP.Q,
                        tTriggerFilterTimeOn:=T#0MS,
                        tTriggerFilterTimeOff:=T#0MS,
                        bWithCapControl:=TRUE,
                      	bNoKeepTryingMove:=FALSE,//bylo true
                        bTriggerCap:=VIS_ROPP.bROPPPuttedCheckOK,
                        bReset:=bResetStates,
                        iEntranceArrayElements:=1,
                        iExitArrayElements:=3,
                        eClearPackageState:=eClearPackageState,
                        eEntranceState:=eBeforeROPPCapControlPackageState,
                        eExitState:=eBeforeROPP2PackageState,
                        bKeepTryingMove:=bKeepTryingMoveROPP2,
						bRFIDReaded:=bRFIDSBeforeROPPWriteToRegister,
                        iBottleWithoutCap:=iROPPFeederCheckCountNOK,
						bError=>,
                        iError=>,
                        bTriggerDone=>,
                        bTriggerFilteredOUT=>);   
				


// --------------------------------------




//Resetowanie
(*IF P00_PackML.rtCycleReseting.Q THEN	
	FOR i := 1 TO 17 DO 
		eBeforeROPPCapControlPackageState[i]	:=		eClearPackageState;
		eBeforeROPPPackageState[i]				:=		eClearPackageState;			
		eBeforeROPP2PackageState[i]				:=		eClearPackageState;		
		eUnderROPPPackageState[i]				:=		eClearPackageState;			
		eUnderROPPCorrectCapPackageState[i]		:=		eClearPackageState;
	END_FOR
END_IF*)
END_ACTION

ACTION aInFormatSensorFilter:
tonFormatSensorOn	(IN	:=	IbFormCheckFormSensor,		PT	:=	T#40MS);//bylo 20, mk bylo 30 19.06.2024
tonFormatSensorOff	(IN	:=	NOT	IbFormCheckFormSensor,	PT	:=	T#40MS);//bylo 30

IF (tonFormatSensorOn.Q) THEN
	bFormatSensor					:=	TRUE;
ELSIF (tonFormatSensorOff.Q) THEN
	bFormatSensor					:=	FALSE;
END_IF

tonBottleSensorOn	(IN	:=	IbBottleInFormCheckBottleSensor,		PT	:=	T#5MS);
tonBottleSensorOff	(IN	:=	NOT	IbBottleInFormCheckBottleSensor,	PT	:=	T#20MS);

IF (tonBottleSensorOn.Q) THEN
	bBottleSensor					:=	TRUE;
ELSIF (tonBottleSensorOff.Q) THEN
	bBottleSensor					:=	FALSE;
END_IF
END_ACTION

ACTION aRFIDRepairOrderCreate:
(*
Nazwa:			aRFIDRepairOrderCreate 
Opis:			Naprawianie błędnych odczytów RFID - tworzenie tabeli kolejności
Wersja:			v0.1
Data:			2022-06-09
Autor:			DP
Urzadzenia:		
Konfiguracja:	
Info:
- na tablice [0] zawsze podawaj ostatni odczytany RFID według kolejności
- ważna jest maksymalna ilość formatek
*)

//Global Presistent:
AbRFIDFormOrder[1];// Globalny rejestr kolejności formatek

//Co kasować po resetach
nRFIDRepairOrderFirstNumber;
iRFIDRepairNumberOfForms :=	48; //bylo 24


(*******Zmiana kolejności formatek pod zakręcarkami*****)
IF rtRFIDRepairToRotate.Q THEN
	 eUnderScrewerPackageState[2].nCardNumber;	//Teoretycznie wystarczy po każdym ruchu ten numer przenosić do góry w tablicy	
	 FOR i:=1 TO 100 DO
		 IF AbRFIDFormOrder[i]		=		eUnderScrewerPackageState[2].nCardNumber THEN
			IF i = 1 THEN
				nRFIDRepairToRotate								:= AbRFIDFormOrder[1];
				nRFIDRepairToRotateBefore						:= AbRFIDFormOrder[iRFIDRepairAddNumber-1];	//-1 bo to numer do którego wpisze w nastepnym cyklu			
				AbRFIDFormOrder[iRFIDRepairAddNumber-1]			:= nRFIDRepairToRotate;
				AbRFIDFormOrder[0]								:= nRFIDRepairToRotate;
				AbRFIDFormOrder[1]								:= nRFIDRepairToRotateBefore;
				iRFIDRepairCount1								:= iRFIDRepairCount1	+	1;				
				EXIT;
			ELSE
				nRFIDRepairToRotate								:= AbRFIDFormOrder[i];
				nRFIDRepairToRotateBefore						:= AbRFIDFormOrder[i-1];
				AbRFIDFormOrder[i-1]							:= nRFIDRepairToRotate; 
				AbRFIDFormOrder[i]								:= nRFIDRepairToRotateBefore;
				iRFIDRepairCount2								:= iRFIDRepairCount2	+	1;	
				EXIT;
			END_IF
		 END_IF 
	 END_FOR
END_IF

						
(*********Dodawanie numerów RFID do tablicy według kolejności odczytywania*******)
(*********************Dodawanie tylko w miejscu przed dozownikami****************)
IF	rtRFIDRepairAddNumber.Q THEN
	//Jeżeli ponownie odczytano pierwszą formatkę to zacznij zapisywać tablice na nowo
	//Odszukaj ten numer znacznika w tablicy i zacznij od niego na nowo zapisywać
	iRFIDRepairCount3								:= iRFIDRepairCount3	+	1;	
	
	//Zapisz numer 
	nBeforeGatePackageState1nCardNumber	:= eBeforeGatePackageState[1].nCardNumber;

	(**** Startowa formatka****)
		//Jeżeli już odczytana została drugi raz
		IF nBeforeGatePackageState1nCardNumber > 0 AND 
			nRFIDRepairOrderFirstNumber = nBeforeGatePackageState1nCardNumber OR
			iRFIDRepairAddNumber >= iRFIDRepairNumberOfForms
		THEN
			FOR	i:=1 TO 100 DO
				IF AbRFIDFormOrder[i] =  nBeforeGatePackageState1nCardNumber	 THEN
					iRFIDRepairAddNumber 				:=	UINT_TO_INT(i);
					bRFIDRepairOrderFirstNumberSaved	:=	TRUE;
					iRFIDRepairCount4					:=	iRFIDRepairCount4	+	1;	
					EXIT;
				END_IF	
			END_FOR
		END_IF	
		//Zapisywanie znacznika pierwszej formatki 										// Zabezpieczenie przed 999
		IF nRFIDRepairOrderFirstNumber = 0 AND nBeforeGatePackageState1nCardNumber > 0 AND nBeforeGatePackageState1nCardNumber < 500 THEN
			nRFIDRepairOrderFirstNumber		:=	nBeforeGatePackageState1nCardNumber;
			iRFIDRepairCount5				:=	iRFIDRepairCount5	+	1;	
		END_IF
	(**** Startowa formatka****)
	
	(***** Dodawanie numeru ***)
	IF nBeforeGatePackageState1nCardNumber > 0 AND nBeforeGatePackageState1nCardNumber < 500 THEN 
		AbRFIDFormOrder[iRFIDRepairAddNumber]	:=	nBeforeGatePackageState1nCardNumber;
		iRFIDRepairAddNumber					:=	iRFIDRepairAddNumber	+	1;
		AbRFIDFormOrder[0]						:=	nBeforeGatePackageState1nCardNumber; //Zawsze do zerowej zapisuj ostatni numer RFID	
		iRFIDRepairCount6						:=	iRFIDRepairCount6	+	1;
	END_IF

	//Jeżeli odczytało drugi raz tą sama formatkę to zacznij od nowa
	IF bRFIDRepairOrderFirstNumberSaved THEN
		nRFIDRepairOrderFirstNumber			:=	AbRFIDFormOrder[1]	; // Ustaw pierwszy numer jako pierwszy w tablicy
	END_IF
END_IF	

// Jezeli bylo 0, nieodczytana RFID 
IF ftRFIDRepairAddNumber.Q AND nBeforeGatePackageState1nCardNumber	=	0 THEN
	iRFIDRepairAddNumber					:=	iRFIDRepairAddNumber	+	1;
	iRFIDRepairCount7						:=	iRFIDRepairCount7	+	1	;
END_IF

(*******Zacznij od nowa jeżeli licznik przekroczył ilość formatek*******)
IF iRFIDRepairAddNumber > 48 THEN
	iRFIDRepairCount8						:= iRFIDRepairCount8	+	1;
END_IF
	
(*****Kasowanie rozkazów****)
IF ftRFIDRepairAddNumber.Q THEN
	bRFIDRepairOrderFirstNumberSaved		:= FALSE;	
END_IF
END_ACTION

ACTION aRFIDRepairOrderSearch:
(*
Nazwa:			aRFIDRepairOrderSearch 
Opis:			Naprawianie błędnych odczytów RFID - szukanie numeru i wpisywanie
Wersja:			v0.1
Data:			2022-06-09
Autor:			DP
Urzadzenia:		
Konfiguracja:	
Info:
- 
*)

iRFIDRepairAddNumber;
//Global Presistent:
AbRFIDFormOrder[1];// Globalny rejestr kolejności formatek
(*** DOZOWNIKI ***)




(****** WAGI *****)
//WAGI 4
IF eWeightPackageState[4].nCardNumber = 0 AND VIS.bWeight4DoWeighting THEN

		IF 	eWeightPackageState[3].nCardNumber > 0	THEN
			FOR	i:=1 TO 100 DO
				IF AbRFIDFormOrder[i] = eWeightPackageState[3].nCardNumber THEN
						IF AbRFIDFormOrder[i+1] > 0 THEN 
							eWeightPackageState[4].nCardNumber				:=	AbRFIDFormOrder[i+1];
							bRFIDRepairChanged								:=  TRUE;
						ELSE //Jeżeli to koniec tablicy to weż zerowy numer
							eWeightPackageState[4].nCardNumber				:=	AbRFIDFormOrder[0];
							bRFIDRepairChanged								:=  TRUE;
						END_IF
						iWeightPackageState43nCardNumberChangeCounter	:=	iWeightPackageState43nCardNumberChangeCounter	+	1;
					EXIT;
				END_IF
			END_FOR
		END_IF	
		(*...dodac z 1 i 2*)	
END_IF
bRFIDRepairChanged									:=  FALSE;

//WAGI 3
IF eWeightPackageState[3].nCardNumber = 0 AND VIS.bWeight3DoWeighting THEN

		IF 	eWeightPackageState[2].nCardNumber > 0	THEN
			FOR	i:=1 TO 100 DO
				IF AbRFIDFormOrder[i] = eWeightPackageState[2].nCardNumber THEN
						IF AbRFIDFormOrder[i+1] > 0 THEN 
							eWeightPackageState[3].nCardNumber				:=	AbRFIDFormOrder[i+1];
							bRFIDRepairChanged								:=  TRUE;						
						ELSE
							eWeightPackageState[3].nCardNumber				:=	AbRFIDFormOrder[0];
							bRFIDRepairChanged								:=  TRUE;			
						END_IF			
						iWeightPackageState32nCardNumberChangeCounter	:=	iWeightPackageState32nCardNumberChangeCounter	+	1;
					EXIT;
				END_IF
				
			END_FOR
		END_IF
		(**)	
END_IF	
bRFIDRepairChanged									:=  FALSE;

//WAGI 2
IF eWeightPackageState[2].nCardNumber = 0 AND VIS.bWeight2DoWeighting THEN

		IF 	eWeightPackageState[1].nCardNumber > 0	THEN
			FOR	i:=1 TO 100 DO
				IF AbRFIDFormOrder[i] = eWeightPackageState[1].nCardNumber THEN
					IF AbRFIDFormOrder[i+1] > 0 THEN 
						eWeightPackageState[2].nCardNumber				:=	AbRFIDFormOrder[i+1];
						bRFIDRepairChanged								:=  TRUE;
					ELSE
						eWeightPackageState[2].nCardNumber				:=	AbRFIDFormOrder[0];
						bRFIDRepairChanged								:=  TRUE;
					END_IF
					iWeightPackageState21nCardNumberChangeCounter	:=	iWeightPackageState21nCardNumberChangeCounter	+	1;
					EXIT;
				END_IF
			END_FOR
		END_IF
		(*dodac z 1 i 4*)	
END_IF		
bRFIDRepairChanged									:=  FALSE;

//WAGI 1
IF eWeightPackageState[1].nCardNumber = 0 AND VIS.bWeight1DoWeighting THEN

		IF 	eWeightPackageState[2].nCardNumber > 0	THEN
			FOR	i:=1 TO 100 DO
				IF AbRFIDFormOrder[i] = eWeightPackageState[2].nCardNumber THEN
					eWeightPackageState[1].nCardNumber				:=	AbRFIDFormOrder[i-1];
					iWeightPackageState12nCardNumberChangeCounter	:=	iWeightPackageState12nCardNumberChangeCounter	+	1;
					bRFIDRepairChanged								:=  TRUE;
					EXIT;
				END_IF
			END_FOR
		END_IF
		(*dodac z 1 i 4*)	
END_IF		
bRFIDRepairChanged									:=  FALSE;

(*
(***** ZAKRECARKI*****)

//Zakrecarka 2
IF eUnderScrewerPackageState[2].nCardNumber = 0 AND P00_PackML.iGripperScrewerCase = 2 THEN
	IF 	eUnderScrewerPackageState[1].nCardNumber > 0	THEN
		FOR	i:=1 TO 100 DO
			IF AbRFIDFormOrder[i] = eUnderScrewerPackageState[1].nCardNumber THEN
				IF AbRFIDFormOrder[i+1] > 0 THEN 
					eUnderScrewerPackageState[2].nCardNumber		:=	AbRFIDFormOrder[i+1];
					bRFIDRepairChanged								:=  TRUE;
				ELSE
					eUnderScrewerPackageState[2].nCardNumber		:=	AbRFIDFormOrder[0];
					bRFIDRepairChanged								:=  TRUE;
				END_IF
				iUnderScrewerPackageState21nCardNumberChangeCounter	:=	iUnderScrewerPackageState21nCardNumberChangeCounter	+	1;
				
				FOR ir3 := 1 TO 100 DO // Sycnhronizacja danych
					 IF eRFID[ir3].nCardNumber	=	eUnderScrewerPackageState[2].nCardNumber THEN
						eRFID[ir3].bFormPresent 		:=	eUnderScrewerPackageState[2].bFormPresent;
						(*Dodatkowy kod jeżeli nasadka została sprawdzona wczesniej niż odczytał czujnik RFID*)
						eRFID[ir3].bCapOK 				:=	eUnderScrewerPackageState[2].bCapOK;		 	
						eRFID[ir3].bCapPutted 			:=	eUnderScrewerPackageState[2].bCapPutted; 	
						eRFID[ir3].bCapChecked			:=	eUnderScrewerPackageState[2].bCapChecked; 	
						IF eUnderScrewerPackageState[2].bCapOK THEN					
							eRFID[ir3].bBottlePresent 	:=	TRUE;						
						END_IF	
						(*Koniec Dodatkowy kod jeżeli nasadka została sprawdzona wczesniej niż odczytał czujnik RFID*)
						eUnderScrewerPackageState[2]	:=	eRFID[ir3];//Zapisywanie tablicy do wglądu w HMI						
					 END_IF
				END_FOR	
				
				EXIT;
			END_IF
		END_FOR
	END_IF
END_IF

//Zakrecarka 1
IF eUnderScrewerPackageState[1].nCardNumber = 0 AND P00_PackML.iGripperScrewerCase = 2 THEN
	IF 	eUnderScrewerPackageState[2].nCardNumber > 0	THEN
		FOR	i:=1 TO 100 DO
			IF AbRFIDFormOrder[i] = eUnderScrewerPackageState[2].nCardNumber THEN
				eUnderScrewerPackageState[1].nCardNumber		:=	AbRFIDFormOrder[i-1];
				bRFIDRepairChanged								:=  TRUE;
		
				iUnderScrewerPackageState12nCardNumberChangeCounter	:=	iUnderScrewerPackageState12nCardNumberChangeCounter	+	1;
				
				FOR ir3 := 1 TO 100 DO // Sycnhronizacja danych
					 IF eRFID[ir3].nCardNumber	=	eUnderScrewerPackageState[1].nCardNumber THEN
						eRFID[ir3].bFormPresent 		:=	eUnderScrewerPackageState[1].bFormPresent;
						(*Dodatkowy kod jeżeli nasadka została sprawdzona wczesniej niż odczytał czujnik RFID*)
						eRFID[ir3].bCapOK 				:=	eUnderScrewerPackageState[1].bCapOK;		 	
						eRFID[ir3].bCapPutted 			:=	eUnderScrewerPackageState[1].bCapPutted; 	
						eRFID[ir3].bCapChecked			:=	eUnderScrewerPackageState[1].bCapChecked; 	
						IF eUnderScrewerPackageState[1].bCapOK THEN					
							eRFID[ir3].bBottlePresent 	:=	TRUE;						
						END_IF	
						(*Koniec Dodatkowy kod jeżeli nasadka została sprawdzona wczesniej niż odczytał czujnik RFID*)
						eUnderScrewerPackageState[1]	:=	eRFID[ir3];//Zapisywanie tablicy do wglądu w HMI						
					 END_IF
				END_FOR	
				
				EXIT;
			END_IF
		END_FOR
	END_IF
END_IF

*)

rtbBottleDragingStationRun(CLK:=VIS.bBottleDragingStationRun);


// pierwsze miejsce przed zakręcarką
IF eBeforeScrewersPackageState[1].nCardNumber = 0 AND rtbBottleDragingStationRun.Q THEN
	IF eBeforeScrewersPackageState[2].nCardNumber > 0	THEN
		FOR	i:=1 TO 100 DO
			IF AbRFIDFormOrder[i] = eBeforeScrewersPackageState[2].nCardNumber THEN
				IF AbRFIDFormOrder[i-1] > 0 THEN 
					eBeforeScrewersPackageState[1].nCardNumber		:=	AbRFIDFormOrder[i-1];
					bRFIDRepairChanged								:=  TRUE;
				END_IF
				
				iUnderScrewerPackageState111nCardNumberChangeCounter	:=	iUnderScrewerPackageState111nCardNumberChangeCounter	+	1;
				
				FOR ir3 := 1 TO 100 DO // Sycnhronizacja danych
					 IF eRFID[ir3].nCardNumber	=	eBeforeScrewersPackageState[1].nCardNumber THEN
						eRFID[ir3].bFormPresent 		:=	eBeforeScrewersPackageState[1].bFormPresent;
						(*Dodatkowy kod jeżeli nasadka została sprawdzona wczesniej niż odczytał czujnik RFID*)
						eRFID[ir3].bCapOK 				:=	eBeforeScrewersPackageState[1].bCapOK;		 	
						eRFID[ir3].bCapPutted 			:=	eBeforeScrewersPackageState[1].bCapPutted; 	
						eRFID[ir3].bCapChecked			:=	eBeforeScrewersPackageState[1].bCapChecked; 	
						IF eBeforeScrewersPackageState[1].bCapOK THEN					
							eRFID[ir3].bBottlePresent 	:=	TRUE;						
						END_IF	
						(*Koniec Dodatkowy kod jeżeli nasadka została sprawdzona wczesniej niż odczytał czujnik RFID*)
						eBeforeScrewersPackageState[1]	:=	eRFID[ir3];//Zapisywanie tablicy do wglądu w HMI						
					 END_IF
				END_FOR	
				
				EXIT;
			END_IF
		END_FOR
	END_IF
END_IF
bRFIDRepairChanged									:=  FALSE;
// Drugie miejsce przed zakręcarką
IF eBeforeScrewersPackageState[2].nCardNumber = 0 AND rtbBottleDragingStationRun.Q THEN
	IF 	eBeforeScrewers2PackageState[1].nCardNumber > 0	THEN
		FOR	i:=1 TO 100 DO
			IF AbRFIDFormOrder[i] = eBeforeScrewers2PackageState[1].nCardNumber THEN
				IF AbRFIDFormOrder[i+1] > 0 THEN 
					eBeforeScrewersPackageState[2].nCardNumber		:=	AbRFIDFormOrder[i-1];
					bRFIDRepairChanged								:=  TRUE;
				ELSE
					eBeforeScrewersPackageState[2].nCardNumber		:=	AbRFIDFormOrder[0];
					bRFIDRepairChanged								:=  TRUE;
				END_IF
				iUnderScrewerPackageState222nCardNumberChangeCounter	:=	iUnderScrewerPackageState222nCardNumberChangeCounter	+	1;
				
				FOR ir3 := 1 TO 100 DO // Sycnhronizacja danych
					 IF eRFID[ir3].nCardNumber	=	eBeforeScrewersPackageState[2].nCardNumber THEN
						eRFID[ir3].bFormPresent 		:=	eBeforeScrewersPackageState[2].bFormPresent;
						(*Dodatkowy kod jeżeli nasadka została sprawdzona wczesniej niż odczytał czujnik RFID*)
						eRFID[ir3].bCapOK 				:=	eBeforeScrewersPackageState[2].bCapOK;		 	
						eRFID[ir3].bCapPutted 			:=	eBeforeScrewersPackageState[2].bCapPutted; 	
						eRFID[ir3].bCapChecked			:=	eBeforeScrewersPackageState[2].bCapChecked; 	
						IF eBeforeScrewersPackageState[2].bCapOK THEN					
							eRFID[ir3].bBottlePresent 	:=	TRUE;						
						END_IF	
						(*Koniec Dodatkowy kod jeżeli nasadka została sprawdzona wczesniej niż odczytał czujnik RFID*)
						eBeforeScrewersPackageState[2]	:=	eRFID[ir3];//Zapisywanie tablicy do wglądu w HMI						
					 END_IF
				END_FOR	
				
				EXIT;
			END_IF
		END_FOR
	END_IF
END_IF
bRFIDRepairChanged									:=  FALSE;
// Trzecie miejsce przed zakręcarką

IF eBeforeScrewers2PackageState[1].nCardNumber = 0 AND rtbBottleDragingStationRun.Q THEN
	IF 	eBeforeScrewersPackageState[2].nCardNumber > 0	THEN
		FOR	i:=1 TO 100 DO
			IF AbRFIDFormOrder[i] = eBeforeScrewersPackageState[2].nCardNumber THEN
				IF AbRFIDFormOrder[i+1] > 0 THEN 
					eBeforeScrewers2PackageState[1].nCardNumber		:=	AbRFIDFormOrder[i+1];
					bRFIDRepairChanged								:=  TRUE;
				//ELSE
				//	eBeforeScrewers2PackageState[1].nCardNumber		:=	AbRFIDFormOrder[0];
				//	bRFIDRepairChanged								:=  TRUE;
				END_IF
				iUnderScrewerPackageState333nCardNumberChangeCounter	:=	iUnderScrewerPackageState333nCardNumberChangeCounter	+	1;
				
				FOR ir3 := 1 TO 100 DO // Sycnhronizacja danych
					 IF eRFID[ir3].nCardNumber	=	eBeforeScrewers2PackageState[1].nCardNumber THEN
						eRFID[ir3].bFormPresent 		:=	eBeforeScrewers2PackageState[1].bFormPresent;
						(*Dodatkowy kod jeżeli nasadka została sprawdzona wczesniej niż odczytał czujnik RFID*)
						eRFID[ir3].bCapOK 				:=	eBeforeScrewers2PackageState[1].bCapOK;		 	
						eRFID[ir3].bCapPutted 			:=	eBeforeScrewers2PackageState[1].bCapPutted; 	
						eRFID[ir3].bCapChecked			:=	eBeforeScrewers2PackageState[1].bCapChecked; 	
						IF eBeforeScrewers2PackageState[1].bCapOK THEN					
							eRFID[ir3].bBottlePresent 	:=	TRUE;						
						END_IF	
						(*Koniec Dodatkowy kod jeżeli nasadka została sprawdzona wczesniej niż odczytał czujnik RFID*)
						eBeforeScrewers2PackageState[1]	:=	eRFID[ir3];//Zapisywanie tablicy do wglądu w HMI						
					 END_IF
				END_FOR	
				
				EXIT;
			END_IF
		END_FOR
	END_IF
END_IF
bRFIDRepairChanged									:=  FALSE;


(*
(**** Naprawa RFID przed dozownikami***)
rtDispencerDragStation(CLK:=VIS.bFormsDragingRightRun OR VIS.bFormsDragingLeftRun);

//Przed dozownikiem 4
IF eDispencersPackageState[4].nCardNumber = 0 AND rtDispencerDragStation.Q THEN

		IF 	eDispencersPackageState[3].nCardNumber > 0	THEN
			FOR	i:=1 TO 100 DO
				IF AbRFIDFormOrder[i] = eDispencersPackageState[3].nCardNumber THEN
						IF AbRFIDFormOrder[i+1] > 0 THEN 
							eDispencersPackageState[4].nCardNumber			:=	AbRFIDFormOrder[i+1];
							bRFIDRepairChanged								:=  TRUE;
						//ELSE //Jeżeli to koniec tablicy to weż zerowy numer
						//	eWeightPackageState[4].nCardNumber				:=	AbRFIDFormOrder[0];
						//	bRFIDRepairChanged								:=  TRUE;
						END_IF
						iDispencerPackageState4nCardNumberChangeCounter	:=	iDispencerPackageState4nCardNumberChangeCounter	+	1;
					EXIT;
				END_IF
			END_FOR
		END_IF	
END_IF
bRFIDRepairChanged									:=  FALSE;

//Przed dozownikiem 3
IF eDispencersPackageState[3].nCardNumber = 0 AND rtDispencerDragStation.Q THEN

		IF 	eDispencersPackageState[2].nCardNumber > 0	THEN
			FOR	i:=1 TO 100 DO
				IF AbRFIDFormOrder[i] = eDispencersPackageState[2].nCardNumber THEN
						IF AbRFIDFormOrder[i+1] > 0 THEN 
							eDispencersPackageState[3].nCardNumber			:=	AbRFIDFormOrder[i+1];
							bRFIDRepairChanged								:=  TRUE;
						//ELSE //Jeżeli to koniec tablicy to weż zerowy numer
						//	eWeightPackageState[4].nCardNumber				:=	AbRFIDFormOrder[0];
						//	bRFIDRepairChanged								:=  TRUE;
						END_IF
						iDispencerPackageState3nCardNumberChangeCounter	:=	iDispencerPackageState3nCardNumberChangeCounter	+	1;
					EXIT;
				END_IF
			END_FOR
		END_IF	
END_IF
bRFIDRepairChanged									:=  FALSE;

//Przed dozownikiem 2
IF eDispencersPackageState[2].nCardNumber = 0 AND rtDispencerDragStation.Q THEN

		IF 	eDispencersPackageState[1].nCardNumber > 0	THEN
			FOR	i:=1 TO 100 DO
				IF AbRFIDFormOrder[i] = eDispencersPackageState[1].nCardNumber THEN
						IF AbRFIDFormOrder[i+1] > 0 THEN 
							eDispencersPackageState[2].nCardNumber			:=	AbRFIDFormOrder[i+1];
							bRFIDRepairChanged								:=  TRUE;
						//ELSE //Jeżeli to koniec tablicy to weż zerowy numer
						//	eWeightPackageState[4].nCardNumber				:=	AbRFIDFormOrder[0];
						//	bRFIDRepairChanged								:=  TRUE;
						END_IF
						iDispencerPackageState2nCardNumberChangeCounter	:=	iDispencerPackageState2nCardNumberChangeCounter	+	1;
					EXIT;
				END_IF
			END_FOR
		END_IF	
END_IF
bRFIDRepairChanged									:=  FALSE;
//Przed dozownikiem 1
IF eDispencersPackageState[1].nCardNumber = 0 AND rtDispencerDragStation.Q THEN

		IF 	eDispencersPackageState[2].nCardNumber > 0	THEN
			FOR	i:=1 TO 100 DO
				IF AbRFIDFormOrder[i] = eDispencersPackageState[2].nCardNumber THEN
						IF AbRFIDFormOrder[i-1] > 0 THEN 
							eDispencersPackageState[2].nCardNumber			:=	AbRFIDFormOrder[i-1];
							bRFIDRepairChanged								:=  TRUE;
						//ELSE //Jeżeli to koniec tablicy to weż zerowy numer
						//	eWeightPackageState[4].nCardNumber				:=	AbRFIDFormOrder[0];
						//	bRFIDRepairChanged								:=  TRUE;
						END_IF
						iDispencerPackageState1nCardNumberChangeCounter	:=	iDispencerPackageState1nCardNumberChangeCounter	+	1;
					EXIT;
				END_IF
			END_FOR
		END_IF	
END_IF
bRFIDRepairChanged									:=  FALSE;



(**** Naprawa pod robotem ***) 
IF eRobotPackageState[1].nCardNumber = 0  THEN

		IF 	eRobotPackageState[2].nCardNumber > 0	THEN
			FOR	i:=1 TO 100 DO
				IF AbRFIDFormOrder[i] = eRobotPackageState[2].nCardNumber THEN
						IF AbRFIDFormOrder[i-1] > 0 THEN 
							eRobotPackageState[1].nCardNumber			:=	AbRFIDFormOrder[i-1];
							bRFIDRepairChanged								:=  TRUE;
						//ELSE //Jeżeli to koniec tablicy to weż zerowy numer
						//	eWeightPackageState[4].nCardNumber				:=	AbRFIDFormOrder[0];
						//	bRFIDRepairChanged								:=  TRUE;
						END_IF
					
				FOR ir3 := 1 TO 100 DO // Sycnhronizacja danych
					 IF eRFID[ir3].nCardNumber	=	eRobotPackageState[1].nCardNumber THEN
							eRobotPackageState[1]	:=	eRFID[ir3];//Zapisywanie tablicy do wglądu w HMI						
					 END_IF
				END_FOR		
						
					iRobotPackageState1nCardNumberChangeCounter	:=	iRobotPackageState1nCardNumberChangeCounter	+	1;
					EXIT;
				END_IF
			END_FOR
		END_IF	
END_IF
bRFIDRepairChanged									:=  FALSE;

*)
END_ACTION

ACTION aRFIDRepairReset:
IF bRFIDRepairReset THEN
	FOR i:=0 TO 100 DO
		AbRFIDFormOrder[i] 				:=	0;
	END_FOR
	bRFIDRepairReset					:=	FALSE;
	nRFIDRepairOrderFirstNumber 		:=	0;
	iRFIDRepairAddNumber				:=	1;
	nBeforeGatePackageState1nCardNumber :=	0;
	iRFIDRepairCount1					:=	0;
	iRFIDRepairCount2					:=	0;
	iRFIDRepairCount3					:=	0;
	iRFIDRepairCount4					:=	0;
	iRFIDRepairCount5					:=	0;
	iRFIDRepairCount6					:=	0;
	
END_IF
END_ACTION

ACTION aRFIDRepairSignals:
fbRFIDRepairFilteredFormsSensorGate(bIn:=IbFormCheckFormSensor,	tFilterTimeOn:=T#30MS,	tFilterTimeOff:=T#5MS);	//musi być szybciej				

rtRFIDRepairAddNumber	(CLK:=	NOT fbRFIDRepairFilteredFormsSensorGate.bOUT,
						Q=>);
						
ftRFIDRepairAddNumber	(CLK:=	eBeforeGatePackageState[1].bFormPresent,
						Q=>);

rtRFIDRepairToRotate 	(CLK:=	P10_GripperScrewer.fbGripperScrewersDragStation.bCycleDone,
						Q=>);
END_ACTION

ACTION aRFIDRepairStatistic:
iRFIDRepairAddNumber; // Zapisze do tego numeru tablicy
nRFIDRepairOrderFirstNumber;	//Pierwsza odczytana formatka

AbRFIDFormOrder[0];

AbRFIDFormOrder[1];
AbRFIDFormOrder[2];
AbRFIDFormOrder[3];
AbRFIDFormOrder[4];
AbRFIDFormOrder[5];
AbRFIDFormOrder[6];
AbRFIDFormOrder[7];
AbRFIDFormOrder[8];
AbRFIDFormOrder[9];
AbRFIDFormOrder[10];
AbRFIDFormOrder[11];
AbRFIDFormOrder[12];
AbRFIDFormOrder[13];
AbRFIDFormOrder[14];
AbRFIDFormOrder[15];
AbRFIDFormOrder[16];
AbRFIDFormOrder[17];
AbRFIDFormOrder[18];
AbRFIDFormOrder[19];
AbRFIDFormOrder[20];
AbRFIDFormOrder[21];
AbRFIDFormOrder[22];
AbRFIDFormOrder[23];
AbRFIDFormOrder[24];
AbRFIDFormOrder[25];
AbRFIDFormOrder[26];
AbRFIDFormOrder[27];
AbRFIDFormOrder[28];
AbRFIDFormOrder[29];
AbRFIDFormOrder[30];
AbRFIDFormOrder[31];
AbRFIDFormOrder[32];
AbRFIDFormOrder[33];
AbRFIDFormOrder[34];
AbRFIDFormOrder[35];
AbRFIDFormOrder[36];
AbRFIDFormOrder[37];
AbRFIDFormOrder[38];
AbRFIDFormOrder[39];
AbRFIDFormOrder[40];
AbRFIDFormOrder[41];
AbRFIDFormOrder[42];
AbRFIDFormOrder[43];
AbRFIDFormOrder[44];
AbRFIDFormOrder[45];
AbRFIDFormOrder[46];
AbRFIDFormOrder[47];
AbRFIDFormOrder[48];
AbRFIDFormOrder[49];
AbRFIDFormOrder[50];
AbRFIDFormOrder[51];
AbRFIDFormOrder[52];
AbRFIDFormOrder[53];
AbRFIDFormOrder[54];
AbRFIDFormOrder[55];
AbRFIDFormOrder[56];
AbRFIDFormOrder[57];
AbRFIDFormOrder[58];
AbRFIDFormOrder[59];
AbRFIDFormOrder[60];
END_ACTION

ACTION aRFIDWarnings:

(*Brak odczytu RFID przed dozownikami*)(*
TimerRFIDDispencersWarning(IN:= 	
								(
									(eBeforeDispencersPackageState[1].bFormPresent AND eBeforeDispencersPackageState[1].nCardNumber = 0)
								OR 	(eBeforeDispencersPackageState[2].bFormPresent AND eBeforeDispencersPackageState[2].nCardNumber = 0)
								OR 	(eBeforeDispencersPackageState[3].bFormPresent AND eBeforeDispencersPackageState[3].nCardNumber = 0) 
								OR	(eBeforeDispencersPackageState[4].bFormPresent AND eBeforeDispencersPackageState[4].nCardNumber = 0)
								)
								AND P00_PackML.tonLongDelayAfterStart60s.Q AND tofCycleExecute.Q AND NOT bDosingTwoPhases (*dwie fazy uzależnione*)
								, PT:=T#500MS); //dodany dozowanie 2 fazwe
//dodany dozowanie 2 fazowe										
TimerRFIDDispencers2PhaseWarning(IN:= 	
								(
									(eBeforeDispencer34PackageState2Phase[1].bFormPresent AND eBeforeDispencer34PackageState2Phase[1].nCardNumber = 0)
								OR 	(eBeforeDispencer34PackageState2Phase[2].bFormPresent AND eBeforeDispencer34PackageState2Phase[2].nCardNumber = 0))
								AND P00_PackML.tonLongDelayAfterStart60s.Q AND tofCycleExecute.Q AND bDosingTwoPhases
								, PT:=T#500MS); 						

rtTimerRFIDDispencerWarning(CLK:=TimerRFIDDispencersWarning.Q OR TimerRFIDDispencers2PhaseWarning.Q);

IF rtTimerRFIDDispencerWarning.Q THEN
		irtTimerRFIDDispencerWarning:=irtTimerRFIDDispencerWarning+1;
END_IF;
				
IF (TimerRFIDDispencersWarning.Q OR TimerRFIDDispencers2PhaseWarning.Q) AND NOT GeneralWarning1[0].bWarning THEN
	GeneralWarning1[0].bWarning										:=TRUE;
	GeneralWarning1[0].udiWarningCode								:=65;
	GeneralWarning1[0].sDescription									:='RFID | Brak odczytu z czujnika przed dozownikami';
ELSIF NOT TimerRFIDDispencersWarning.Q AND GeneralWarning1[0].bAcknowledge THEN
	GeneralWarning1[0].bWarning										:=FALSE;
	GeneralWarning1[0].bAcknowledge									:=FALSE;
	VIS.uliWarningAcknowledge.6 									:=FALSE;
ELSIF GeneralWarning1[0].bAcknowledge THEN
	GeneralWarning1[0].bAcknowledge									:=TRUE;
END_IF


(*Brak odczytu RFID przed waga*)
TimerRFIDWeightWarning(IN:= 		
								(
									(eWeightPackageState[1].bFormPresent AND eWeightPackageState[1].nCardNumber = 0)
								OR 	(eWeightPackageState[2].bFormPresent AND eWeightPackageState[2].nCardNumber = 0)
								OR 	(eWeightPackageState[3].bFormPresent AND eWeightPackageState[3].nCardNumber = 0) 
								OR	(eWeightPackageState[4].bFormPresent AND eWeightPackageState[4].nCardNumber = 0)
								)
								AND P00_PackML.tonLongDelayAfterStart60s.Q AND tofCycleExecute.Q
								, PT:=T#500MS);
								
IF TimerRFIDWeightWarning.Q AND NOT GeneralWarning1[1].bWarning THEN
	GeneralWarning1[1].bWarning										:=TRUE;
	GeneralWarning1[1].udiWarningCode								:=66;
	GeneralWarning1[1].sDescription									:='RFID | Brak odczytu z czujnika przed wagami';
ELSIF NOT TimerRFIDWeightWarning.Q AND GeneralWarning1[1].bAcknowledge THEN
	GeneralWarning1[1].bWarning										:=FALSE;
	GeneralWarning1[1].bAcknowledge									:=FALSE;
	VIS.uliWarningAcknowledge.7 									:=FALSE;
ELSIF GeneralWarning1[1].bAcknowledge THEN
	GeneralWarning1[1].bAcknowledge									:=TRUE;
END_IF


(*Brak odczytu RFID przed zakrecarka*)
eBeforeScrewers2PackageState[2].nID; eBeforeScrewers2PackageState[2].nCardNumber; eBeforeScrewers2PackageState[2].bFormPresent;
eBeforeScrewers2PackageState[1].nID; eBeforeScrewers2PackageState[1].nCardNumber; eBeforeScrewers2PackageState[1].bFormPresent;
eBeforeScrewersPackageState[2].nID; eBeforeScrewersPackageState[2].nCardNumber; eBeforeScrewersPackageState[2].bFormPresent; 
eBeforeScrewersPackageState[1].nID; eBeforeScrewersPackageState[1].nCardNumber; eBeforeScrewersPackageState[1].bFormPresent; 
//[1..3] Struktura pod zakręcarkami                                                                                     
eUnderScrewerPackageState[2].nID; eUnderScrewerPackageState[2].nCardNumber; eUnderScrewerPackageState[2].bFormPresent; 
eUnderScrewerPackageState[1].nID; eUnderScrewerPackageState[1].nCardNumber; eUnderScrewerPackageState[1].bFormPresent; 
// [1..12] Struktura za zakręcarkami                                                                                   
eAfterScrewerPackageState[2].nID; eAfterScrewerPackageState[2].nCardNumber; eAfterScrewerPackageState[2].bFormPresent; 
eAfterScrewerPackageState[1].nID; eAfterScrewerPackageState[1].nCardNumber; eAfterScrewerPackageState[1].bFormPresent; 

TimerRFIDScrewersWarning(IN:=	   
								(	
									(eBeforeScrewers2PackageState[1].bFormPresent	AND eBeforeScrewers2PackageState[1].nCardNumber = 0)
								OR (eBeforeScrewers2PackageState[2].bFormPresent	AND eBeforeScrewers2PackageState[2].nCardNumber = 0)
								OR (eBeforeScrewersPackageState[2].bFormPresent 	AND eBeforeScrewersPackageState[2].nCardNumber = 0)
								OR (eBeforeScrewersPackageState[1].bFormPresent 	AND eBeforeScrewersPackageState[1].nCardNumber = 0)
								)
								AND P00_PackML.tonLongDelayAfterStart60s.Q AND tofCycleExecute.Q
								, PT:=T#500MS);
			
								
								
rtTimerRFIDScrewersWarning	(CLK:=TimerRFIDScrewersWarning.Q, Q=>);

IF rtTimerRFIDScrewersWarning.Q THEN
	irtTimerRFIDScrewersWarning := irtTimerRFIDScrewersWarning + 1;
END_IF

IF TimerRFIDScrewersWarning.Q AND NOT GeneralWarning1[2].bWarning THEN
	GeneralWarning1[2].bWarning										:=TRUE;
	GeneralWarning1[2].udiWarningCode								:=67;
	GeneralWarning1[2].sDescription									:='RFID | Brak odczytu z czujnika przed zakręcarką';
ELSIF NOT TimerRFIDScrewersWarning.Q AND GeneralWarning1[2].bAcknowledge THEN
	GeneralWarning1[2].bWarning										:=FALSE;
	GeneralWarning1[2].bAcknowledge									:=FALSE;
	VIS.uliWarningAcknowledge.8 									:=FALSE;
ELSIF GeneralWarning1[2].bAcknowledge THEN
	GeneralWarning1[2].bAcknowledge									:=TRUE;
END_IF


(*Brak odczytu RFID pod robotem*)
(*TimerRFIDRobotWarning(IN:=
								(
						 			(eRobotPackageState[1].bFormPresent AND eRobotPackageState[1].nCardNumber = 0)
								OR	(eRobotPackageState[2].bFormPresent AND eRobotPackageState[2].nCardNumber = 0)
								)
								AND P00_PackML.tonLongDelayAfterStart60s.Q AND tofCycleExecute.Q
								,PT:=T#500MS);*)
								
IF TimerRFIDRobotWarning.Q AND NOT GeneralWarning1[3].bWarning THEN
	GeneralWarning1[3].bWarning										:=TRUE;
	GeneralWarning1[3].udiWarningCode								:=68;
	GeneralWarning1[3].sDescription									:='RFID | Brak odczytu z czujnika przed robotem';
ELSIF NOT TimerRFIDRobotWarning.Q AND GeneralWarning1[3].bAcknowledge THEN
	GeneralWarning1[3].bWarning										:=FALSE;
	GeneralWarning1[3].bAcknowledge									:=FALSE;
	VIS.uliWarningAcknowledge.9 									:=FALSE;
ELSIF GeneralWarning1[3].bAcknowledge THEN
	GeneralWarning1[3].bAcknowledge									:=TRUE;
END_IF*)
END_ACTION

ACTION aScope:
//Przeciąganie pod zakręcarkami
//Wszystkie potrzebne zmienne do wykresów

MAIN.IbBottleInFormCheckBottleSensor;
MAIN.IbFormCheckFormSensor;
VIS.bGateBeforeDispencersRun;
P00_ReadRFIDCard.bReadedCardDispencer;

MAIN.IbFourthFormCheckFormSensor;
MAIN.IbSecondFormCheckFormSensor;

VIS.bFormsDragingLeftRun;
VIS.bFormsDragingRightRun;
eBeforeDispencersPackageState[1].bFormPresent;
eBeforeDispencersPackageState[2].bFormPresent;
eBeforeDispencersPackageState[3].bFormPresent;
eBeforeDispencersPackageState[4].bFormPresent;
eDispencersPackageState[1].bFormPresent;
eDispencersPackageState[2].bFormPresent;
eDispencersPackageState[3].bFormPresent;
eDispencersPackageState[4].bFormPresent;

iFormsDragingFormCounter;
P02_Dispencers.fbDispencersDragLeftStation.eRunningState;

//Przeciąganie pod robotem
//Wszystkie potrzebne zmienne do wykresów
eRobotPackageState[1].bFormPresent;
eRobotPackageState[2].bFormPresent;
P13_BottleTransfer.IbFirstFormCheckFormSensor;
P13_BottleTransfer.IbSecondFormCheckFormSensor;
P00_PackML.iBottleTransferCase;
P00_PackML.iRobotPickCase;
P00_PackML.nCounterForms;
P00_PackML.nCounterFormsToLoad;
VIS.bGateRobotEntranceRun;
bRobotStationDone;
VIS.bBottleTransferRun;
P13_BottleTransfer.IbBottleCheckAfterBottleTransferSensor;
END_ACTION

ACTION aSetIDBottle:
(*
Nazwa:			aSetIDBottle 
Opis:			Nadawanie ID butelką
Wersja:			v0.1
Data:			2018-10-10
Autor:			DP
Urzadzenia:		
Konfiguracja:	
Info:
*)


rtBeforeGateDispencerStateNotPresent(CLK:=eBeforeGatePackageState[1].bFormPresent, Q=>);
rtBeforeGateDispencerFormPresent(CLK:= Main.IbFormCheckFormSensor);

IF rtBeforeGateDispencerFormPresent.Q THEN
		eBeforeGatePackageState[1].bFormPresent :=TRUE;
 		eBeforeGatePackageState[1].nID := nID + 1 ;
		nID:= eBeforeGatePackageState[1].nID ;
END_IF

// Zapisywanie obecności butelki pod podjanikiem butelek

rtibBottleFeederrFormPresent(CLK:=fbIbBottleFeederFormPresent.bOUT);

IF rtibBottleFeederrFormPresent.Q THEN
	eBottleFeederPackageState[1].bFormPresent :=TRUE;
END_IF
END_ACTION

ACTION aSimulation:
rtSimulationSetRegisters(CLK:=VIS.bSimulation AND NOT P13_BottleTransfer.IbFirstFormCheckFormSensor,Q=>);




(*Sumulacja*) 
	IF rtSimulationSetRegisters.Q THEN
		bSimulationForLoop:=TRUE;
	END_IF

IF bSimulationForLoop THEN
	FOR is := 1 TO 100 DO	
		IF nSimulationCardNumber = eRFID[is].nCardNumber THEN	//Jeżeli znaleziono w tablicy takie RFID 
			eRFID[is].bBottlePresent	:= 	TRUE;
			eRFID[is].nDispencerNr		:=  iCountSimulation;
			IF iCountSimulation=5 THEN	eRFID[is].bWeightOK 			:= 	FALSE;	ELSE;	eRFID[is].bWeightOK 			:= TRUE;	END_IF;      
			IF iCountSimulation=50 THEN	eRFID[is].bWeightTooLow 		:= 	TRUE;	ELSE;	eRFID[is].bWeightTooLow 		:= FALSE;	END_IF;   
			IF iCountSimulation=100 THEN	eRFID[is].bWeightTooHigh		:= 	TRUE;	ELSE;	eRFID[is].bWeightTooHigh		:= FALSE;	END_IF;   
			IF iCountSimulation=150 THEN	eRFID[is].bCapOK 				:= 	FALSE;	ELSE 	eRFID[is].bCapOK 				:= TRUE;	END_IF;        
			IF iCountSimulation=200 THEN	eRFID[is].bCapGripperScrewed	:= 	FALSE;	ELSE 	eRFID[is].bCapGripperScrewed	:= TRUE;	eRFID[is].bCapGripperScrewAborted	:= FALSE;	END_IF;
			IF iCountSimulation=250 THEN	eRFID[is].bCapCorrectNOK		:= 	TRUE;	ELSE 	eRFID[is].bCapCorrectNOK		:= FALSE;	END_IF;   
			IF iCountSimulation=300 THEN	eRFID[is].bCapCorrectCapOn 		:= 	FALSE;	ELSE 	eRFID[is].bCapCorrectCapOn 		:= TRUE;	END_IF;
			iCountSimulation			:= iCountSimulation +1 ;
		END_IF
		
		bSimulationForLoop := FALSE;
	END_FOR	
END_IF

	
	IF 	iCountSimulation	>	1000 THEN
		iCountSimulation := 0;
	END_IF
END_ACTION

ACTION aStartingPoint:
(*
Nazwa:			aStartingPoint 
Opis:			Stan początkowy maszyny
Wersja:			v0.2
Data:			2022-02-01
Autor:			DJ
Urzadzenia:		
Konfiguracja:	
Info:
*)

// Nowe zmienne reset	
	eBeforeDispencer12PackageState2Phase[1]			:=eClearPackageState;	
	eBeforeDispencer12PackageState2Phase[2]         :=eClearPackageState;
	eBeforeDispencer34PackageState2Phase[1]	        :=eClearPackageState;
	eBeforeDispencer34PackageState2Phase[2]	        :=eClearPackageState;
	eBeforeDispencer12PackageState2Phase[1].bFormPresent	:=	TRUE;
	eBeforeDispencer12PackageState2Phase[2].bFormPresent	:=	TRUE;
	eBeforeDispencer34PackageState2Phase[1].bFormPresent	:=	TRUE;
	eBeforeDispencer34PackageState2Phase[2].bFormPresent	:=	TRUE;
	eBeforeDispencer12PackageState2Phase[1].nCardNumber 	:= 	999; //Przypisanie po resecie, żeby robot nie pobierał butelki i ostrzezenie sie nie wyświetlało
	eBeforeDispencer12PackageState2Phase[2].nCardNumber 	:= 	999; //Przypisanie po resecie, żeby robot nie pobierał butelki i ostrzezenie sie nie wyświetlało
	eBeforeDispencer34PackageState2Phase[2].nCardNumber 	:= 	999; //Przypisanie po resecie, żeby robot nie pobierał butelki i ostrzezenie sie nie wyświetlało
	eBeforeDispencer34PackageState2Phase[1].nCardNumber 	:= 	999; //Przypisanie po resecie, żeby robot nie pobierał butelki i ostrzezenie sie nie wyświetlało

	
	eDispencer12PackageState2Phase[1]				:=eClearPackageState;      
	eDispencer12PackageState2Phase[2]       		:=eClearPackageState;
	eDispencer34PackageState2Phase[1]       		:=eClearPackageState;
	eDispencer34PackageState2Phase[2]       		:=eClearPackageState;
		
	eDispencer12PackageState2Phase[1].bFormPresent	:=	TRUE;//TRUE;
	eDispencer12PackageState2Phase[2].bFormPresent	:=	TRUE;	
	eDispencer34PackageState2Phase[1].bFormPresent	:=	TRUE;//TRUE;
	eDispencer34PackageState2Phase[2].bFormPresent	:=	TRUE;	

	eDispencer12PackageState2Phase[1].nCardNumber	:=	999;//TRUE;
	eDispencer12PackageState2Phase[2].nCardNumber	:=	999;	
	eDispencer34PackageState2Phase[1].nCardNumber	:=	999;//TRUE;
	eDispencer34PackageState2Phase[2].nCardNumber	:=	999;	

	
	

	eAfterDispencer12PackageState2Phase[1]				:=eClearPackageState;
	eAfterDispencer12PackageState2Phase[2]				:=eClearPackageState;
	eAfterDispencer34PackageState2Phase[1]				:=eClearPackageState;
	eAfterDispencer34PackageState2Phase[2]				:=eClearPackageState;
	
	eAfterDispencer12PackageState2Phase[1].bFormPresent	:=	FALSE;
	eAfterDispencer12PackageState2Phase[2].bFormPresent	:=	FALSE;
	eAfterDispencer34PackageState2Phase[1].bFormPresent	:=	FALSE;
	eAfterDispencer34PackageState2Phase[2].bFormPresent	:=	FALSE;
	
	
	

	eWeightPackage2PhasePackageState[2].bFormPresent		:=	FALSE;
	eWeightPackage2PhasePackageState[1].bFormPresent		:=	FALSE;
	

	eBeforeGatePackageState[1].bFormPresent			:=	TRUE;
	eBeforeGatePackageState[1].	nCardNumber 		:=	999; //Przypisanie po resecie, żeby robot nie pobierał butelki i ostrzezenie sie nie wyświetlało
	
	eBeforeDispencersPackageState[4].bFormPresent	:=	TRUE;
	eBeforeDispencersPackageState[3].bFormPresent	:=	TRUE;
	eBeforeDispencersPackageState[2].bFormPresent	:=	TRUE;
	eBeforeDispencersPackageState[1].bFormPresent	:=	TRUE;
	eBeforeDispencersPackageState[4].nCardNumber 	:= 	999; //Przypisanie po resecie, żeby robot nie pobierał butelki i ostrzezenie sie nie wyświetlało
	eBeforeDispencersPackageState[3].nCardNumber 	:= 	999; //Przypisanie po resecie, żeby robot nie pobierał butelki i ostrzezenie sie nie wyświetlało
	eBeforeDispencersPackageState[2].nCardNumber 	:= 	999; //Przypisanie po resecie, żeby robot nie pobierał butelki i ostrzezenie sie nie wyświetlało
	eBeforeDispencersPackageState[1].nCardNumber 	:= 	999; //Przypisanie po resecie, żeby robot nie pobierał butelki i ostrzezenie sie nie wyświetlało
	
	FOR id:=1 TO 4 DO
		eDispencersPackageState[id].bFormPresent	:=	FALSE;//TRUE;
	END_FOR			
	FOR ia:=1 TO 4 DO	
		eAfterDispencersPackageState[ia].bFormPresent:=	FALSE;
	END_FOR
	FOR iw:=1 TO 5 DO	
		eWeightPackageState[iw].bFormPresent		:=	FALSE;
	END_FOR
	
	eBeforeScrewers2PackageState[2].bFormPresent	:=	TRUE;
	eBeforeScrewers2PackageState[1].bFormPresent	:=	TRUE;
	eBeforeScrewersPackageState[2].bFormPresent		:=	TRUE;
	eBeforeScrewersPackageState[1].bFormPresent		:=	TRUE;
	eBeforeScrewers2PackageState[2].nCardNumber 	:= 	999; //Przypisanie po resecie, żeby robot nie pobierał butelki i ostrzezenie sie nie wyświetlało
	eBeforeScrewers2PackageState[1].nCardNumber 	:= 	999; //Przypisanie po resecie, żeby robot nie pobierał butelki i ostrzezenie sie nie wyświetlało
	eBeforeScrewersPackageState[2].nCardNumber 		:= 	999; //Przypisanie po resecie, żeby robot nie pobierał butelki i ostrzezenie sie nie wyświetlało
	eBeforeScrewersPackageState[1].nCardNumber 		:= 	999; //Przypisanie po resecie, żeby robot nie pobierał butelki i ostrzezenie sie nie wyświetlało
	
	
	eUnderScrewerPackageState[1]					:=eClearPackageState;
	eUnderScrewerPackageState[2]					:=eClearPackageState;	
	eUnderScrewerPackageState[1].bFormPresent		:=TRUE;
	eUnderScrewerPackageState[2].bFormPresent		:=TRUE;	
	
	
	//eRobotPackageState[1].bFormPresent				:=	TRUE; 
	//eRobotPackageState[2].bFormPresent				:=	TRUE;
	//eRobotPackageState[1].nCardNumber 				:= 	999; //Przypisanie po resecie, żeby robot nie pobierał butelki i ostrzezenie sie nie wyświetlało
   // eRobotPackageState[2].nCardNumber 				:= 	999; //Przypisanie po resecie, żeby robot nie pobierał butelki i ostrzezenie sie nie wyświetlało
	
	eRobotTempState[1]:=eClearPackageState; //testy 31.05
END_ACTION

ACTION aStatistics:
(*
Nazwa:			aStatistics 
Opis:			Podgląd rejestrów formatek
Wersja:			v0.1
Data:			2018-10-10
Autor:			DP
Urzadzenia:		
Konfiguracja:	
Info:
*)
// podajnik butelek
P01_BottleFeeder.fbBottleFeeder.tCycleTime;
//łapanie szyjki
P02_Dispencers.fbDispencersCatch1Station.eRunningState;
P02_Dispencers.fbDispencersCatch2Station.eRunningState;
P02_Dispencers.fbDispencersCatch3Station.eRunningState;
P02_Dispencers.fbDispencersCatch4Station.eRunningState;
//Cykl pracy Dozowniki
P02_Dispencers.fbDispencer1.tCycleTime;
P02_Dispencers.fbDispencer2.tCycleTime;
P02_Dispencers.fbDispencer3.tCycleTime;
P02_Dispencers.fbDispencer4.tCycleTime;
P02_Dispencers.fbDispencersCatch1Station.tCycleTime;
P02_Dispencers.fbDispencersCatch2Station.tCycleTime;
P02_Dispencers.fbDispencersCatch3Station.tCycleTime;
P02_Dispencers.fbDispencersCatch4Station.tCycleTime;


//Cykl Przesuwania formatek
P02_Dispencers.fbDispencersDragLeftStation.tCycleTime;
P02_Dispencers.fbDispencersDragRightStation.tCycleTime;
//Cykl pracy wagi
P05_Weight.fbWeight1.tCycleTime;
P05_Weight.fbWeight2.tCycleTime;
P05_Weight.fbWeight3.tCycleTime;
P05_Weight.fbWeight4.tCycleTime;

//Cykl sprawdzania 
P09_CapPuttedCheck.fbCapPuttedCheck.tCycleTime;

//Cykl pod zakręcarkami

P10_GripperScrewer.fb2GripperScrewer1.tCycleTime;
P10_GripperScrewer.fb2GripperScrewer2.tCycleTime;
P10_GripperScrewer.fbGripperScrewer1CatchStation.tCycleTime;
P10_GripperScrewer.fbGripperScrewer2CatchStation.tCycleTime;

P10_GripperScrewer.fbGripperScrewersDragStation.tCycleTime;


P13_BottleTransfer.fbBottleTransfer.tCycleTime;

// [1.......2] Strukutira pod podajnikiem
eBottleFeederPackageState[1].bFormPresent; eBottleFeederPackageState[1].bBottlePresent; 





eBeforeGatePackageState[1].bFormPresent; eBeforeGatePackageState[1].bBottlePresent; eBeforeGatePackageState[1].nCardNumber;


// [1..1] Struktura przed dozownikami przed szlabanem
eBeforeDispencersPackageState[4].bFormPresent; eBeforeDispencersPackageState[4].bBottlePresent; eBeforeDispencersPackageState[4].nID; eBeforeDispencersPackageState[4].nCardNumber;
eBeforeDispencersPackageState[3].bFormPresent; eBeforeDispencersPackageState[3].bBottlePresent; eBeforeDispencersPackageState[3].nID; eBeforeDispencersPackageState[3].nCardNumber;
eBeforeDispencersPackageState[2].bFormPresent; eBeforeDispencersPackageState[2].bBottlePresent; eBeforeDispencersPackageState[2].nID; eBeforeDispencersPackageState[2].nCardNumber;
eBeforeDispencersPackageState[1].bFormPresent; eBeforeDispencersPackageState[1].bBottlePresent; eBeforeDispencersPackageState[1].nID; eBeforeDispencersPackageState[1].nCardNumber;


// [1..4] Struktura pod dozownikami
eDispencersPackageState[4].nID; eDispencersPackageState[4].nCardNumber; eDispencersPackageState[4].bFormPresent; eDispencersPackageState[4].bBottlePresent; eDispencersPackageState[4].bDosingTwoPhases; eDispencersPackageState[4].lrDoseVolumeSV; eDispencersPackageState[4].lrDoseVolumeSVSecondPhase;  eDispencersPackageState[4].lrDoseVolumeCV; eDispencersPackageState[4].lrDoseVolumeCVSecondPhase; eDispencersPackageState[4].nDispencerNr; eDispencersPackageState[4].nDispencerNrSecondPhase; eDispencersPackageState[4].tDispencingTime; eDispencersPackageState[4].tDispencingTimeSecondPhase; 
eDispencersPackageState[3].nID; eDispencersPackageState[3].nCardNumber; eDispencersPackageState[3].bFormPresent; eDispencersPackageState[3].bBottlePresent; eDispencersPackageState[3].bDosingTwoPhases; eDispencersPackageState[3].lrDoseVolumeSV; eDispencersPackageState[3].lrDoseVolumeSVSecondPhase;  eDispencersPackageState[3].lrDoseVolumeCV; eDispencersPackageState[3].lrDoseVolumeCVSecondPhase; eDispencersPackageState[3].nDispencerNr; eDispencersPackageState[3].nDispencerNrSecondPhase; eDispencersPackageState[3].tDispencingTime; eDispencersPackageState[3].tDispencingTimeSecondPhase;
eDispencersPackageState[2].nID; eDispencersPackageState[2].nCardNumber; eDispencersPackageState[2].bFormPresent; eDispencersPackageState[2].bBottlePresent; eDispencersPackageState[2].bDosingTwoPhases; eDispencersPackageState[2].lrDoseVolumeSV; eDispencersPackageState[2].lrDoseVolumeSVSecondPhase;  eDispencersPackageState[2].lrDoseVolumeCV; eDispencersPackageState[2].lrDoseVolumeCVSecondPhase; eDispencersPackageState[2].nDispencerNr; eDispencersPackageState[2].nDispencerNrSecondPhase; eDispencersPackageState[2].tDispencingTime; eDispencersPackageState[2].tDispencingTimeSecondPhase;
eDispencersPackageState[1].nID; eDispencersPackageState[1].nCardNumber; eDispencersPackageState[1].bFormPresent; eDispencersPackageState[1].bBottlePresent; eDispencersPackageState[1].bDosingTwoPhases; eDispencersPackageState[1].lrDoseVolumeSV; eDispencersPackageState[1].lrDoseVolumeSVSecondPhase;  eDispencersPackageState[1].lrDoseVolumeCV; eDispencersPackageState[1].lrDoseVolumeCVSecondPhase; eDispencersPackageState[1].nDispencerNr; eDispencersPackageState[1].nDispencerNrSecondPhase; eDispencersPackageState[1].tDispencingTime; eDispencersPackageState[1].tDispencingTimeSecondPhase;

// [1..4] Struktura za dozownikami i przed wagą	
eAfterDispencersPackageState[4].nID; eAfterDispencersPackageState[4].nCardNumber; eAfterDispencersPackageState[4].bFormPresent; eAfterDispencersPackageState[4].bBottlePresent; eAfterDispencersPackageState[4].bDosingTwoPhases; eAfterDispencersPackageState[4].lrDoseVolumeSV; eAfterDispencersPackageState[4].lrDoseVolumeSVSecondPhase;  eAfterDispencersPackageState[4].lrDoseVolumeCV; eAfterDispencersPackageState[4].lrDoseVolumeCVSecondPhase; eAfterDispencersPackageState[4].nDispencerNr; eAfterDispencersPackageState[4].nDispencerNrSecondPhase; eAfterDispencersPackageState[4].tDispencingTime; eAfterDispencersPackageState[4].tDispencingTimeSecondPhase; 
eAfterDispencersPackageState[3].nID; eAfterDispencersPackageState[3].nCardNumber; eAfterDispencersPackageState[3].bFormPresent; eAfterDispencersPackageState[3].bBottlePresent; eAfterDispencersPackageState[3].bDosingTwoPhases; eAfterDispencersPackageState[3].lrDoseVolumeSV; eAfterDispencersPackageState[3].lrDoseVolumeSVSecondPhase;  eAfterDispencersPackageState[3].lrDoseVolumeCV; eAfterDispencersPackageState[3].lrDoseVolumeCVSecondPhase; eAfterDispencersPackageState[3].nDispencerNr; eAfterDispencersPackageState[3].nDispencerNrSecondPhase; eAfterDispencersPackageState[3].tDispencingTime; eAfterDispencersPackageState[3].tDispencingTimeSecondPhase; 
eAfterDispencersPackageState[2].nID; eAfterDispencersPackageState[2].nCardNumber; eAfterDispencersPackageState[2].bFormPresent; eAfterDispencersPackageState[2].bBottlePresent; eAfterDispencersPackageState[2].bDosingTwoPhases; eAfterDispencersPackageState[2].lrDoseVolumeSV; eAfterDispencersPackageState[2].lrDoseVolumeSVSecondPhase;  eAfterDispencersPackageState[2].lrDoseVolumeCV; eAfterDispencersPackageState[2].lrDoseVolumeCVSecondPhase; eAfterDispencersPackageState[2].nDispencerNr; eAfterDispencersPackageState[2].nDispencerNrSecondPhase; eAfterDispencersPackageState[2].tDispencingTime; eAfterDispencersPackageState[2].tDispencingTimeSecondPhase; 
eAfterDispencersPackageState[1].nID; eAfterDispencersPackageState[1].nCardNumber; eAfterDispencersPackageState[1].bFormPresent; eAfterDispencersPackageState[1].bBottlePresent; eAfterDispencersPackageState[1].bDosingTwoPhases; eAfterDispencersPackageState[1].lrDoseVolumeSV; eAfterDispencersPackageState[1].lrDoseVolumeSVSecondPhase;  eAfterDispencersPackageState[1].lrDoseVolumeCV; eAfterDispencersPackageState[1].lrDoseVolumeCVSecondPhase; eAfterDispencersPackageState[1].nDispencerNr; eAfterDispencersPackageState[1].nDispencerNrSecondPhase; eAfterDispencersPackageState[1].tDispencingTime; eAfterDispencersPackageState[1].tDispencingTimeSecondPhase; 

//////////////////////////////////////////
// Struktura dla 2fazy
// Struktura przed dozownikami 2 faza 
eBeforeDispencer12PackageState2Phase[2].bFormPresent; eBeforeDispencer12PackageState2Phase[2].bBottlePresent; eBeforeDispencer12PackageState2Phase[2].nID; eBeforeDispencer12PackageState2Phase[2].nCardNumber;
eBeforeDispencer12PackageState2Phase[1].bFormPresent; eBeforeDispencer12PackageState2Phase[1].bBottlePresent; eBeforeDispencer12PackageState2Phase[1].nID; eBeforeDispencer12PackageState2Phase[1].nCardNumber;
// pierwsza faza
eBeforeDispencer34PackageState2Phase[2].bFormPresent; eBeforeDispencer34PackageState2Phase[2].bBottlePresent; eBeforeDispencer34PackageState2Phase[2].nID; eBeforeDispencer34PackageState2Phase[2].nCardNumber;
eBeforeDispencer34PackageState2Phase[1].bFormPresent; eBeforeDispencer34PackageState2Phase[1].bBottlePresent; eBeforeDispencer34PackageState2Phase[1].nID; eBeforeDispencer34PackageState2Phase[1].nCardNumber;

// [1..2] Struktura za dozownikami i przed wagą	dwufazowe
eAfterDispencer12PackageState2Phase[2].nID; eAfterDispencer12PackageState2Phase[2].nCardNumber; eAfterDispencer12PackageState2Phase[2].bFormPresent; eAfterDispencer12PackageState2Phase[2].bBottlePresent; eAfterDispencer12PackageState2Phase[2].bDosingTwoPhases; eAfterDispencer12PackageState2Phase[2].lrDoseVolumeSV; eAfterDispencer12PackageState2Phase[2].lrDoseVolumeSVSecondPhase;  eAfterDispencer12PackageState2Phase[2].lrDoseVolumeCV; eAfterDispencer12PackageState2Phase[2].lrDoseVolumeCVSecondPhase; eAfterDispencer12PackageState2Phase[2].nDispencerNr; eAfterDispencer12PackageState2Phase[2].nDispencerNrSecondPhase; eAfterDispencer12PackageState2Phase[2].tDispencingTime; eAfterDispencer12PackageState2Phase[2].tDispencingTimeSecondPhase; 
eAfterDispencer12PackageState2Phase[1].nID; eAfterDispencer12PackageState2Phase[1].nCardNumber; eAfterDispencer12PackageState2Phase[1].bFormPresent; eAfterDispencer12PackageState2Phase[1].bBottlePresent; eAfterDispencer12PackageState2Phase[1].bDosingTwoPhases; eAfterDispencer12PackageState2Phase[1].lrDoseVolumeSV; eAfterDispencer12PackageState2Phase[1].lrDoseVolumeSVSecondPhase;  eAfterDispencer12PackageState2Phase[1].lrDoseVolumeCV; eAfterDispencer12PackageState2Phase[1].lrDoseVolumeCVSecondPhase; eAfterDispencer12PackageState2Phase[1].nDispencerNr; eAfterDispencer12PackageState2Phase[1].nDispencerNrSecondPhase; eAfterDispencer12PackageState2Phase[1].tDispencingTime; eAfterDispencer12PackageState2Phase[1].tDispencingTimeSecondPhase; 
// [1..2] Struktura za dozownikami 34 - pierwsza faza
eAfterDispencer34PackageState2Phase[2].nID; eAfterDispencer34PackageState2Phase[2].nCardNumber; eAfterDispencer34PackageState2Phase[2].bFormPresent; eAfterDispencer34PackageState2Phase[2].bBottlePresent; eAfterDispencer34PackageState2Phase[2].bDosingTwoPhases; eAfterDispencer34PackageState2Phase[2].lrDoseVolumeSV; eAfterDispencer34PackageState2Phase[2].lrDoseVolumeSVSecondPhase;  eAfterDispencer34PackageState2Phase[2].lrDoseVolumeCV; eAfterDispencer34PackageState2Phase[2].lrDoseVolumeCVSecondPhase; eAfterDispencer34PackageState2Phase[2].nDispencerNr; eAfterDispencer34PackageState2Phase[2].nDispencerNrSecondPhase; eAfterDispencer34PackageState2Phase[2].tDispencingTime; eAfterDispencer34PackageState2Phase[2].tDispencingTimeSecondPhase; 
eAfterDispencer34PackageState2Phase[1].nID; eAfterDispencer34PackageState2Phase[1].nCardNumber; eAfterDispencer34PackageState2Phase[1].bFormPresent; eAfterDispencer34PackageState2Phase[1].bBottlePresent; eAfterDispencer34PackageState2Phase[1].bDosingTwoPhases; eAfterDispencer34PackageState2Phase[1].lrDoseVolumeSV; eAfterDispencer34PackageState2Phase[1].lrDoseVolumeSVSecondPhase;  eAfterDispencer34PackageState2Phase[1].lrDoseVolumeCV; eAfterDispencer34PackageState2Phase[1].lrDoseVolumeCVSecondPhase; eAfterDispencer34PackageState2Phase[1].nDispencerNr; eAfterDispencer34PackageState2Phase[1].nDispencerNrSecondPhase; eAfterDispencer34PackageState2Phase[1].tDispencingTime; eAfterDispencer34PackageState2Phase[1].tDispencingTimeSecondPhase; 

// dozowniki
// [1..2] Struktura pod dozownikami
eDispencer12PackageState2Phase[2].nID; eDispencer12PackageState2Phase[2].nCardNumber; eDispencer12PackageState2Phase[2].bFormPresent; eDispencer12PackageState2Phase[2].bBottlePresent; eDispencer12PackageState2Phase[2].bDosingTwoPhases; eDispencer12PackageState2Phase[2].lrDoseVolumeSV; eDispencer12PackageState2Phase[2].lrDoseVolumeSVSecondPhase;  eDispencer12PackageState2Phase[2].lrDoseVolumeCV; eDispencer12PackageState2Phase[2].lrDoseVolumeCVSecondPhase; eDispencer12PackageState2Phase[2].nDispencerNr; eDispencer12PackageState2Phase[2].nDispencerNrSecondPhase; eDispencer12PackageState2Phase[2].tDispencingTime; eDispencer12PackageState2Phase[2].tDispencingTimeSecondPhase;
eDispencer12PackageState2Phase[1].nID; eDispencer12PackageState2Phase[1].nCardNumber; eDispencer12PackageState2Phase[1].bFormPresent; eDispencer12PackageState2Phase[1].bBottlePresent; eDispencer12PackageState2Phase[1].bDosingTwoPhases; eDispencer12PackageState2Phase[1].lrDoseVolumeSV; eDispencer12PackageState2Phase[1].lrDoseVolumeSVSecondPhase;  eDispencer12PackageState2Phase[1].lrDoseVolumeCV; eDispencer12PackageState2Phase[1].lrDoseVolumeCVSecondPhase; eDispencer12PackageState2Phase[1].nDispencerNr; eDispencer12PackageState2Phase[1].nDispencerNrSecondPhase; eDispencer12PackageState2Phase[1].tDispencingTime; eDispencer12PackageState2Phase[1].tDispencingTimeSecondPhase;

eDispencer34PackageState2Phase[2].nID; eDispencer34PackageState2Phase[2].nCardNumber; eDispencer34PackageState2Phase[2].bFormPresent; eDispencer34PackageState2Phase[2].bBottlePresent; eDispencer34PackageState2Phase[2].bDosingTwoPhases; eDispencer34PackageState2Phase[2].lrDoseVolumeSV; eDispencer34PackageState2Phase[2].lrDoseVolumeSVSecondPhase;  eDispencer34PackageState2Phase[2].lrDoseVolumeCV; eDispencer34PackageState2Phase[2].lrDoseVolumeCVSecondPhase; eDispencer34PackageState2Phase[2].nDispencerNr; eDispencer34PackageState2Phase[2].nDispencerNrSecondPhase; eDispencer34PackageState2Phase[2].tDispencingTime; eDispencer34PackageState2Phase[2].tDispencingTimeSecondPhase;
eDispencer34PackageState2Phase[1].nID; eDispencer34PackageState2Phase[1].nCardNumber; eDispencer34PackageState2Phase[1].bFormPresent; eDispencer34PackageState2Phase[1].bBottlePresent; eDispencer34PackageState2Phase[1].bDosingTwoPhases; eDispencer34PackageState2Phase[1].lrDoseVolumeSV; eDispencer34PackageState2Phase[1].lrDoseVolumeSVSecondPhase;  eDispencer34PackageState2Phase[1].lrDoseVolumeCV; eDispencer34PackageState2Phase[1].lrDoseVolumeCVSecondPhase; eDispencer34PackageState2Phase[1].nDispencerNr; eDispencer34PackageState2Phase[1].nDispencerNrSecondPhase; eDispencer34PackageState2Phase[1].tDispencingTime; eDispencer34PackageState2Phase[1].tDispencingTimeSecondPhase;


